KUKA KRL program: MyProgram_069().src

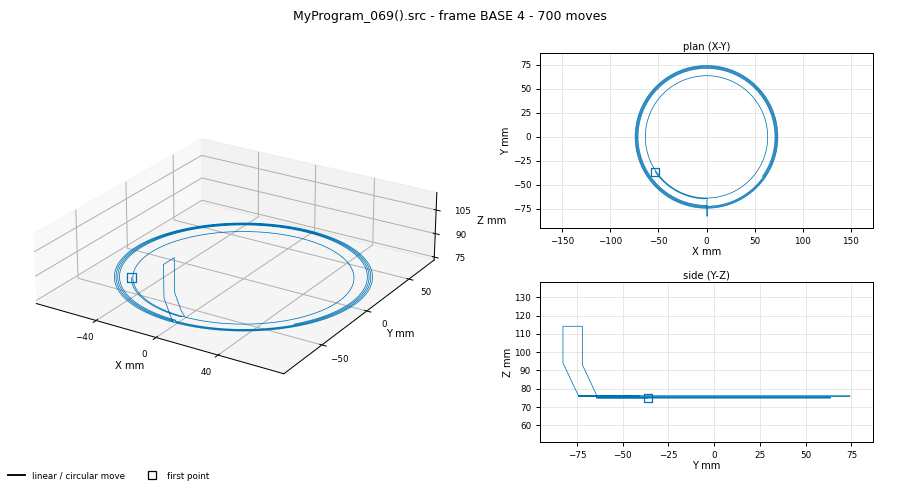
[picture p0: tool path of MyProgram_069().src in frame BASE 4, 700 of 700 moves have a stored position in this frame; points joined in program order, loops and branches not executed]
&ACCESS RVP
&REL 1
&PARAM TEMPLATE = C:\KRC\Roboter\Template\vorgabe
&PARAM EDITMASK = *
DEF MyProgram_069()
; ---- Setting reference (Base) ----
$BASE = BASE_DATA[4]

; --------------------------
; ---- Setting tool (TCP) ----
$TOOL = TOOL_DATA[3]
; --------------------------

$VEL.CP = VEL_APROX_PRINT
Startdeposition()
$VEL.CP = VEL_PRINT
LIN {X -53.2736,Y -36.3857,Z 75,A -150.3803,B 24.8918,C -2.4023,E1 24.8694,E2 -125.5307} C_DIS
LIN {X -51.112,Y -39.3636,Z 75,A -147.7583,B 24.8936,C -2.3813,E1 24.8737,E2 -128.1152} C_DIS
LIN {X -49.4525,Y -41.43,Z 75,A -144.3336,B 24.8921,C -2.3979,E1 24.8799,E2 -131.5953} C_DIS
LIN {X -46.3505,Y -44.8729,Z 75,A -140.9445,B 24.8943,C -2.3739,E1 24.8863,E2 -134.942} C_DIS
LIN {X -44.9329,Y -46.2927,Z 75,A -138.7085,B 24.8937,C -2.3797,E1 24.8908,E2 -137.2012} C_DIS
LIN {X -41.3789,Y -49.495,Z 75,A -134.5886,B 24.8947,C -2.3689,E1 24.8995,E2 -141.3115} C_DIS
LIN {X -38.5752,Y -51.7101,Z 75,A -131.7311,B 24.8958,C -2.3566,E1 24.9058,E2 -144.1501} C_DIS
LIN {X -36.3603,Y -53.2908,Z 75,A -129.2902,B 24.8961,C -2.3532,E1 24.9113,E2 -146.5913} C_DIS
LIN {X -34.0806,Y -54.7764,Z 75,A -126.7495,B 24.8961,C -2.3522,E1 24.9174,E2 -149.1377} C_DIS
LIN {X -31.5265,Y -56.2851,Z 75,A -124.1519,B 24.8966,C -2.3478,E1 24.9236,E2 -151.7325} C_DIS
LIN {X -29.0657,Y -57.5953,Z 75,A -121.6814,B 24.8969,C -2.3445,E1 24.9298,E2 -154.202} C_DIS
LIN {X -26.5923,Y -58.7774,Z 75,A -118.8897,B 24.8964,C -2.3496,E1 24.9369,E2 -157.0127} C_DIS
LIN {X -23.076,Y -60.2452,Z 75,A -115.9709,B 24.8976,C -2.3361,E1 24.9444,E2 -159.9057} C_DIS
LIN {X -20.7754,Y -61.0765,Z 75,A -113.7684,B 24.8977,C -2.335,E1 24.9502,E2 -162.1098} C_DIS
LIN {X -18.3054,Y -61.8615,Z 75,A -111.6866,B 24.8983,C -2.3285,E1 24.9557,E2 -164.1797} C_DIS
LIN {X -16.0814,Y -62.4765,Z 75,A -109.3686,B 24.8979,C -2.3332,E1 24.962,E2 -166.5126} C_DIS
LIN {X -13.5706,Y -63.0698,Z 75,A -107.0172,B 24.8979,C -2.3335,E1 24.9684,E2 -168.8676} C_DIS
LIN {X -10.8355,Y -63.5969,Z 75,A -104.5216,B 24.8979,C -2.3331,E1 24.9753,E2 -171.3649} C_DIS
LIN {X -7.9994,Y -64.0158,Z 75,A -102.109,B 24.8982,C -2.3296,E1 24.9819,E2 -173.771} C_DIS
LIN {X -4.131,Y -64.381,Z 75,A -98.8452,B 24.8986,C -2.3252,E1 24.991,E2 -177.0258} C_DIS
LIN {X -2.1333,Y -64.4779,Z 75,A -96.0689,B 24.8965,C -2.3486,E1 24.9989,E2 -179.8581} C_DIS
LIN {X -2.1333,Y -64.4779,Z 75,A -96.0689,B 24.8965,C -2.3486,E1 24.9989,E2 -179.8581} C_DIS
Enddeposition()
LIN {X 0.4536,Y -63.6088,Z 75,A -94.8897,B 24.8974,C -2.3386,E1 25.0022,E2 -181.0136} C_DIS
Startdeposition()
$VEL.CP = VEL_PRINT
LIN {X -1.5862,Y -63.5949,Z 75,A -97.6108,B 24.8992,C -2.3183,E1 24.9944,E2 -178.2442} C_DIS
LIN {X -4.665,Y -63.4434,Z 75,A -100.413,B 24.8992,C -2.3176,E1 24.9866,E2 -175.4395} C_DIS
LIN {X -7.7944,Y -63.1354,Z 75,A -103.2285,B 24.8992,C -2.3183,E1 24.9788,E2 -172.6239} C_DIS
LIN {X -10.8862,Y -62.6763,Z 75,A -106.0478,B 24.8991,C -2.319,E1 24.971,E2 -169.8036} C_DIS
LIN {X -13.9401,Y -62.0686,Z 75,A -108.8562,B 24.8991,C -2.3201,E1 24.9633,E2 -166.9946} C_DIS
LIN {X -16.9609,Y -61.312,Z 75,A -111.6742,B 24.8989,C -2.3215,E1 24.9557,E2 -164.1756} C_DIS
LIN {X -19.9607,Y -60.402,Z 75,A -114.4932,B 24.8987,C -2.3237,E1 24.9482,E2 -161.3568} C_DIS
LIN {X -22.895,Y -59.352,Z 75,A -117.3072,B 24.8985,C -2.326,E1 24.9408,E2 -158.5426} C_DIS
LIN {X -25.7932,Y -58.151,Z 75,A -120.1357,B 24.8982,C -2.3289,E1 24.9336,E2 -155.7143} C_DIS
LIN {X -28.6026,Y -56.8219,Z 75,A -122.9457,B 24.898,C -2.332,E1 24.9265,E2 -152.9043} C_DIS
LIN {X -31.3638,Y -55.3457,Z 75,A -125.7172,B 24.8975,C -2.3367,E1 24.9197,E2 -150.1363} C_DIS
LIN {X -33.5624,Y -54.0396,Z 75,A -128.0227,B 24.8973,C -2.34,E1 24.9143,E2 -147.8315} C_DIS
LIN {X -36.0815,Y -52.3917,Z 75,A -130.7821,B 24.897,C -2.3433,E1 24.9078,E2 -145.0708} C_DIS
LIN {X -38.5515,Y -50.6023,Z 75,A -133.5526,B 24.8966,C -2.3475,E1 24.9016,E2 -142.3004} C_DIS
LIN {X -40.9565,Y -48.6766,Z 75,A -136.3489,B 24.8962,C -2.3522,E1 24.8956,E2 -139.5047} C_DIS
LIN {X -43.2647,Y -46.6366,Z 75,A -139.132,B 24.8957,C -2.3574,E1 24.8898,E2 -136.7229} C_DIS
LIN {X -45.4504,Y -44.5087,Z 75,A -141.8393,B 24.8951,C -2.3639,E1 24.8845,E2 -134.0197} C_DIS
LIN {X -47.4246,Y -42.3981,Z 75,A -144.3013,B 24.8944,C -2.3724,E1 24.8799,E2 -131.567} C_DIS
LIN {X -49.1892,Y -40.3391,Z 75,A -146.9641,B 24.8943,C -2.3736,E1 24.8751,E2 -128.8949} C_DIS
LIN {X -51.0948,Y -37.8967,Z 75,A -149.7751,B 24.8937,C -2.3799,E1 24.8703,E2 -126.0854} C_DIS
LIN {X -52.8961,Y -35.339,Z 75,A -152.6098,B 24.8931,C -2.3865,E1 24.8658,E2 -123.2525} C_DIS
LIN {X -54.5639,Y -32.7051,Z 75,A -155.4478,B 24.8925,C -2.3932,E1 24.8617,E2 -120.416} C_DIS
LIN {X -56.1094,Y -29.9761,Z 75,A -158.2749,B 24.8918,C -2.4007,E1 24.8579,E2 -117.5918} C_DIS
LIN {X -57.5088,Y -27.1951,Z 75,A -161.0971,B 24.8912,C -2.408,E1 24.8544,E2 -114.7719} C_DIS
LIN {X -58.7706,Y -24.3485,Z 75,A -163.9365,B 24.8905,C -2.4153,E1 24.8513,E2 -111.9341} C_DIS
LIN {X -59.8972,Y -21.4281,Z 75,A -166.7555,B 24.8898,C -2.4234,E1 24.8486,E2 -109.1187} C_DIS
LIN {X -60.8747,Y -18.4692,Z 75,A -169.5856,B 24.8891,C -2.4313,E1 24.8462,E2 -106.291} C_DIS
LIN {X -61.7097,Y -15.4515,Z 75,A -172.4241,B 24.8883,C -2.4394,E1 24.8441,E2 -103.4554} C_DIS
LIN {X -62.3925,Y -12.4103,Z 75,A -175.2521,B 24.8876,C -2.4475,E1 24.8425,E2 -100.6303} C_DIS
LIN {X -62.9255,Y -9.3393,Z 75,A -178.0797,B 24.8868,C -2.4558,E1 24.8413,E2 -97.8057} C_DIS
LIN {X -63.3083,Y -6.237,Z 75,A 179.0777,B 24.886,C -2.4641,E1 24.8404,E2 -94.9658} C_DIS
LIN {X -63.5384,Y -3.1165,Z 75,A 176.2485,B 24.8852,C -2.4727,E1 24.8399,E2 -92.1403} C_DIS
LIN {X -63.6159,Y -0.0035,Z 75,A 173.3835,B 24.8845,C -2.4805,E1 24.8398,E2 -89.2765} C_DIS
LIN {X -63.5377,Y 3.1302,Z 75,A 170.5787,B 24.8836,C -2.4898,E1 24.8401,E2 -86.4771} C_DIS
LIN {X -63.3082,Y 6.2374,Z 75,A 167.7516,B 24.8828,C -2.4983,E1 24.8408,E2 -83.6533} C_DIS
LIN {X -62.9269,Y 9.3298,Z 75,A 164.9241,B 24.882,C -2.5067,E1 24.8418,E2 -80.8291} C_DIS
LIN {X -62.3946,Y 12.3995,Z 75,A 162.0978,B 24.8813,C -2.5152,E1 24.8433,E2 -78.0062} C_DIS
LIN {X -61.7084,Y 15.4568,Z 75,A 159.2405,B 24.8805,C -2.5233,E1 24.8451,E2 -75.1517} C_DIS
LIN {X -60.8705,Y 18.4828,Z 75,A 156.41,B 24.8796,C -2.532,E1 24.8473,E2 -72.3256} C_DIS
LIN {X -59.894,Y 21.4369,Z 75,A 153.5875,B 24.8789,C -2.5402,E1 24.8498,E2 -69.5067} C_DIS
LIN {X -58.774,Y 24.3404,Z 75,A 150.763,B 24.8781,C -2.5483,E1 24.8528,E2 -66.6855} C_DIS
LIN {X -57.5134,Y 27.1852,Z 75,A 147.9417,B 24.8773,C -2.5562,E1 24.856,E2 -63.8678} C_DIS
LIN {X -56.2186,Y 29.7687,Z 75,A 145.5305,B 24.8763,C -2.5674,E1 24.8591,E2 -61.4704} C_DIS
LIN {X -54.9606,Y 32.0339,Z 75,A 142.9607,B 24.876,C -2.5695,E1 24.8627,E2 -58.8924} C_DIS
LIN {X -53.3179,Y 34.6991,Z 75,A 140.1379,B 24.8753,C -2.5773,E1 24.8669,E2 -56.0738} C_DIS
LIN {X -51.5598,Y 37.2616,Z 75,A 137.3184,B 24.8746,C -2.5845,E1 24.8714,E2 -53.2575} C_DIS
LIN {X -49.8386,Y 39.5325,Z 75,A 134.7611,B 24.8739,C -2.5914,E1 24.8758,E2 -50.7046} C_DIS
LIN {X -47.895,Y 41.866,Z 75,A 131.9989,B 24.8733,C -2.5978,E1 24.8808,E2 -47.9451} C_DIS
LIN {X -45.8014,Y 44.1466,Z 75,A 129.1848,B 24.8727,C -2.6041,E1 24.8861,E2 -45.1338} C_DIS
LIN {X -43.5781,Y 46.3427,Z 75,A 126.4974,B 24.8718,C -2.6131,E1 24.8915,E2 -42.4568} C_DIS
LIN {X -41.5304,Y 48.1876,Z 75,A 123.8613,B 24.8715,C -2.6157,E1 24.897,E2 -39.8163} C_DIS
LIN {X -39.1322,Y 50.1548,Z 75,A 121.052,B 24.871,C -2.6213,E1 24.9032,E2 -37.0101} C_DIS
LIN {X -36.6395,Y 52.0036,Z 75,A 118.2409,B 24.8705,C -2.6266,E1 24.9095,E2 -34.2018} C_DIS
LIN {X -34.0348,Y 53.7445,Z 75,A 115.4063,B 24.87,C -2.6317,E1 24.9161,E2 -31.3701} C_DIS
LIN {X -31.3169,Y 55.372,Z 75,A 112.5717,B 24.8694,C -2.6371,E1 24.923,E2 -28.5398} C_DIS
LIN {X -28.5819,Y 56.8322,Z 75,A 109.7423,B 24.869,C -2.6409,E1 24.93,E2 -25.7118} C_DIS
LIN {X -25.7746,Y 58.1593,Z 75,A 106.934,B 24.8686,C -2.6449,E1 24.9371,E2 -22.9059} C_DIS
LIN {X -22.9048,Y 59.3481,Z 75,A 104.1261,B 24.8683,C -2.6484,E1 24.9444,E2 -20.1004} C_DIS
LIN {X -19.9491,Y 60.4059,Z 75,A 101.3458,B 24.8679,C -2.6528,E1 24.9517,E2 -17.3253} C_DIS
LIN {X -17.5047,Y 61.158,Z 75,A 99.0947,B 24.8675,C -2.6564,E1 24.9577,E2 -15.0789} C_DIS
LIN {X -14.6786,Y 61.898,Z 75,A 96.3519,B 24.8675,C -2.6566,E1 24.9651,E2 -12.3326} C_DIS
LIN {X -11.6341,Y 62.5418,Z 75,A 93.5368,B 24.8673,C -2.6586,E1 24.9729,E2 -9.5191} C_DIS
LIN {X -9.1143,Y 62.9575,Z 75,A 91.3179,B 24.8669,C -2.6619,E1 24.979,E2 -7.3062} C_DIS
LIN {X -6.1891,Y 63.3127,Z 75,A 88.5793,B 24.8669,C -2.6615,E1 24.9866,E2 -4.5649} C_DIS
LIN {X -3.0984,Y 63.5392,Z 75,A 85.7848,B 24.8669,C -2.6625,E1 24.9944,E2 -1.772} C_DIS
LIN {X 0.0032,Y 63.6148,Z 75,A 82.9856,B 24.8669,C -2.6631,E1 25.0022,E2 1.026} C_DIS
LIN {X 3.1338,Y 63.5375,Z 75,A 80.1649,B 24.8669,C -2.6633,E1 25.01,E2 3.8456} C_DIS
LIN {X 6.2357,Y 63.3084,Z 75,A 77.3535,B 24.8669,C -2.6629,E1 25.0179,E2 6.6563} C_DIS
LIN {X 9.3404,Y 62.9253,Z 75,A 74.5461,B 24.8669,C -2.6624,E1 25.0256,E2 9.4624} C_DIS
LIN {X 12.4092,Y 62.3927,Z 75,A 71.7413,B 24.8669,C -2.6614,E1 25.0333,E2 12.2666} C_DIS
LIN {X 15.4667,Y 61.7059,Z 75,A 68.9232,B 24.8671,C -2.6599,E1 25.041,E2 15.0841} C_DIS
LIN {X 18.47,Y 60.8744,Z 75,A 66.1206,B 24.8673,C -2.6581,E1 25.0485,E2 17.8864} C_DIS
LIN {X 21.4292,Y 59.8968,Z 75,A 63.3044,B 24.8676,C -2.6555,E1 25.0559,E2 20.7031} C_DIS
LIN {X 24.3533,Y 58.7686,Z 75,A 60.5053,B 24.8678,C -2.6533,E1 25.0632,E2 23.5012} C_DIS
LIN {X 27.1924,Y 57.5101,Z 75,A 57.7015,B 24.8681,C -2.6499,E1 25.0703,E2 26.3058} C_DIS
LIN {X 29.9949,Y 56.0994,Z 75,A 54.8938,B 24.8685,C -2.6467,E1 25.0773,E2 29.1134} C_DIS
LIN {X 32.706,Y 54.5633,Z 75,A 52.0953,B 24.8688,C -2.6429,E1 25.084,E2 31.9123} C_DIS
LIN {X 35.3388,Y 52.8962,Z 75,A 49.3009,B 24.8692,C -2.6389,E1 25.0906,E2 34.7072} C_DIS
LIN {X 37.8864,Y 51.1024,Z 75,A 46.4928,B 24.8697,C -2.6341,E1 25.0969,E2 37.5168} C_DIS
LIN {X 40.3605,Y 49.1718,Z 75,A 43.6883,B 24.8702,C -2.6294,E1 25.103,E2 40.3217} C_DIS
LIN {X 42.7186,Y 47.1377,Z 75,A 40.8915,B 24.8707,C -2.6242,E1 25.1089,E2 43.12} C_DIS
LIN {X 44.9873,Y 44.9775,Z 75,A 38.0869,B 24.8712,C -2.6188,E1 25.1145,E2 45.9256} C_DIS
LIN {X 47.1345,Y 42.7221,Z 75,A 35.2939,B 24.8718,C -2.6129,E1 25.1198,E2 48.7202} C_DIS
LIN {X 49.1744,Y 40.3574,Z 75,A 32.4874,B 24.8724,C -2.6066,E1 25.1249,E2 51.5287} C_DIS
LIN {X 51.1003,Y 37.8892,Z 75,A 29.6918,B 24.873,C -2.6005,E1 25.1296,E2 54.3256} C_DIS
LIN {X 52.8943,Y 35.3417,Z 75,A 27.0861,B 24.8732,C -2.5984,E1 25.1337,E2 56.9234} C_DIS
LIN {X 54.1864,Y 33.3262,Z 75,A 24.7652,B 24.8742,C -2.5888,E1 25.1372,E2 59.2552} C_DIS
LIN {X 55.742,Y 30.6537,Z 75,A 21.9932,B 24.8749,C -2.5818,E1 25.141,E2 62.0296} C_DIS
LIN {X 57.1695,Y 27.9014,Z 75,A 19.2132,B 24.8756,C -2.5744,E1 25.1445,E2 64.8121} C_DIS
LIN {X 58.4611,Y 25.0825,Z 75,A 16.4284,B 24.8763,C -2.5668,E1 25.1476,E2 67.5998} C_DIS
LIN {X 59.6287,Y 22.1644,Z 75,A 13.623,B 24.877,C -2.5593,E1 25.1505,E2 70.4073} C_DIS
LIN {X 60.6496,Y 19.1951,Z 75,A 10.8159,B 24.8778,C -2.5515,E1 25.1529,E2 73.217} C_DIS
LIN {X 61.5159,Y 16.2058,Z 75,A 8.0311,B 24.8785,C -2.5436,E1 25.155,E2 76.0046} C_DIS
LIN {X 62.2351,Y 13.1768,Z 75,A 5.2439,B 24.8793,C -2.5354,E1 25.1567,E2 78.7948} C_DIS
LIN {X 62.8086,Y 10.0955,Z 75,A 2.6298,B 24.8797,C -2.532,E1 25.158,E2 81.4017} C_DIS
LIN {X 63.1502,Y 7.6694,Z 75,A 0.2777,B 24.8807,C -2.5215,E1 25.1588,E2 83.7648} C_DIS
LIN {X 63.4448,Y 4.6442,Z 75,A -2.4543,B 24.8815,C -2.513,E1 25.1595,E2 86.5005} C_DIS
LIN {X 63.5907,Y 1.723,Z 75,A -5.0784,B 24.8822,C -2.505,E1 25.1598,E2 89.128} C_DIS
LIN {X 63.5948,Y -1.5886,Z 75,A -8.0424,B 24.8831,C -2.496,E1 25.1597,E2 92.0957} C_DIS
LIN {X 63.4416,Y -4.6895,Z 75,A -10.82,B 24.8838,C -2.4876,E1 25.1592,E2 94.8766} C_DIS
LIN {X 63.1371,Y -7.7813,Z 75,A -13.6018,B 24.8846,C -2.4791,E1 25.1583,E2 97.6619} C_DIS
LIN {X 62.6766,Y -10.885,Z 75,A -16.4077,B 24.8854,C -2.4707,E1 25.1571,E2 100.4712} C_DIS
LIN {X 62.0686,Y -13.9403,Z 75,A -19.1944,B 24.8862,C -2.4624,E1 25.1555,E2 103.2614} C_DIS
LIN {X 61.3116,Y -16.9624,Z 75,A -21.9821,B 24.887,C -2.4541,E1 25.1535,E2 106.0527} C_DIS
LIN {X 60.4077,Y -19.9434,Z 75,A -24.7683,B 24.8877,C -2.4459,E1 25.1512,E2 108.8423} C_DIS
LIN {X 59.3578,Y -22.8796,Z 75,A -27.5816,B 24.8885,C -2.4373,E1 25.1484,E2 111.6604} C_DIS
LIN {X 58.1492,Y -25.7973,Z 75,A -30.3781,B 24.8892,C -2.4299,E1 25.1453,E2 114.4589} C_DIS
LIN {X 56.8221,Y -28.6023,Z 75,A -33.159,B 24.8899,C -2.4221,E1 25.1419,E2 117.2435} C_DIS
LIN {X 55.3471,Y -31.3614,Z 75,A -35.9584,B 24.8906,C -2.4144,E1 25.1382,E2 120.0464} C_DIS
LIN {X 53.7461,Y -34.0323,Z 75,A -38.7473,B 24.8913,C -2.4069,E1 25.1341,E2 122.8388} C_DIS
LIN {X 52.3355,Y -36.1624,Z 75,A -40.9259,B 24.8916,C -2.4037,E1 25.1307,E2 125.0143} C_DIS
LIN {X 50.616,Y -38.5337,Z 75,A -43.653,B 24.8924,C -2.3944,E1 25.1261,E2 127.7503} C_DIS
LIN {X 48.6741,Y -40.9594,Z 75,A -46.4378,B 24.893,C -2.3875,E1 25.1212,E2 130.5385} C_DIS
LIN {X 46.6155,Y -43.2878,Z 75,A -49.2468,B 24.8937,C -2.3802,E1 25.1159,E2 133.3523} C_DIS
LIN {X 44.4109,Y -45.5466,Z 75,A -52.0468,B 24.8942,C -2.3745,E1 25.1104,E2 136.154} C_DIS
LIN {X 42.1345,Y -47.6605,Z 75,A -54.8314,B 24.8947,C -2.3684,E1 25.1046,E2 138.9419} C_DIS
LIN {X 39.7565,Y -49.6614,Z 75,A -57.6197,B 24.8953,C -2.3625,E1 25.0986,E2 141.7334} C_DIS
LIN {X 37.2535,Y -51.5656,Z 75,A -60.4288,B 24.8957,C -2.3572,E1 25.0923,E2 144.5449} C_DIS
LIN {X 34.6862,Y -53.3264,Z 75,A -63.2303,B 24.8962,C -2.3518,E1 25.0858,E2 147.3498} C_DIS
LIN {X 32.0353,Y -54.9598,Z 75,A -66.0387,B 24.8967,C -2.3466,E1 25.079,E2 150.162} C_DIS
LIN {X 29.2897,Y -56.4708,Z 75,A -68.8327,B 24.897,C -2.3425,E1 25.0721,E2 152.9576} C_DIS
LIN {X 26.5014,Y -57.8317,Z 75,A -71.621,B 24.8974,C -2.3383,E1 25.0651,E2 155.7487} C_DIS
LIN {X 23.8555,Y -58.9714,Z 75,A -73.967,B 24.8972,C -2.3405,E1 25.0591,E2 158.0841} C_DIS
LIN {X 21.4149,Y -59.9018,Z 75,A -76.5529,B 24.898,C -2.3319,E1 25.0523,E2 160.685} C_DIS
LIN {X 18.4567,Y -60.8784,Z 75,A -79.3518,B 24.8982,C -2.3287,E1 25.0448,E2 163.4861} C_DIS
LIN {X 15.4544,Y -61.709,Z 75,A -81.9653,B 24.8982,C -2.3303,E1 25.0378,E2 166.0918} C_DIS
LIN {X 13.1313,Y -62.2445,Z 75,A -84.2896,B 24.8986,C -2.3243,E1 25.0314,E2 168.4273} C_DIS
LIN {X 10.0828,Y -62.8105,Z 75,A -87.0793,B 24.8988,C -2.3222,E1 25.0237,E2 171.219} C_DIS
LIN {X 7.0055,Y -63.2278,Z 75,A -89.8194,B 24.8988,C -2.3217,E1 25.0161,E2 173.958} C_DIS
LIN {X 4.4282,Y -63.4594,Z 75,A -92.137,B 24.8989,C -2.3209,E1 25.0097,E2 176.2763} C_DIS
LIN {X 1.4801,Y -63.5971,Z 75,A -94.8431,B 24.8991,C -2.319,E1 25.0021,E2 178.9864} C_DIS
LIN {X 1.4801,Y -63.5971,Z 75,A -94.8431,B 24.8991,C -2.319,E1 25.0021,E2 178.9864} C_DIS
Enddeposition()
LIN {X 0.4776,Y -65.7217,Z 79.5315,A -94.88,B 24.8977,C -2.3345,E1 25.0021,E2 178.9864} C_DIS
LIN {X 0.5496,Y -72.0606,Z 93.1262,A -94.8556,B 24.8986,C -2.3242,E1 25.0021,E2 178.9864} C_DIS
LIN {X 0.5496,Y -72.0606,Z 114.1262,A -95.2134,B 24.885,C -2.4748,E1 25.0021,E2 178.9864} C_DIS
LIN {X 0.6266,Y -82.6562,Z 114.1262,A -94.6615,B 24.9002,C -2.3061,E1 25.0026,E2 178.8353} C_DIS
LIN {X 0.6266,Y -82.6562,Z 94.1262,A -94.3209,B 24.9123,C -2.1627,E1 25.0026,E2 178.8353} C_DIS
LIN {X 0.5379,Y -76.3176,Z 80.5315,A -94.3434,B 24.9115,C -2.1722,E1 25.0026,E2 178.8353} C_DIS
LIN {X 0.5083,Y -74.2047,Z 76,A -94.3524,B 24.9112,C -2.176,E1 25.0026,E2 178.8353} C_DIS
Startdeposition()
$VEL.CP = VEL_PRINT
LIN {X 3.1308,Y -74.1412,Z 76,A -92.2496,B 24.911,C -2.1787,E1 25.0084,E2 176.7265} C_DIS
LIN {X 5.9684,Y -73.9669,Z 76,A -90.1014,B 24.911,C -2.1785,E1 25.0144,E2 174.5799} C_DIS
LIN {X 8.5765,Y -73.71,Z 76,A -88.0356,B 24.9108,C -2.1808,E1 25.0202,E2 172.51} C_DIS
LIN {X 11.2837,Y -73.3444,Z 76,A -85.9296,B 24.9107,C -2.1821,E1 25.026,E2 170.4027} C_DIS
LIN {X 14.0849,Y -72.8583,Z 76,A -83.5817,B 24.9102,C -2.1881,E1 25.0325,E2 168.0433} C_DIS
LIN {X 17.1465,Y -72.2006,Z 76,A -81.2572,B 24.9102,C -2.1877,E1 25.0388,E2 165.7228} C_DIS
LIN {X 19.9124,Y -71.4865,Z 76,A -79.0131,B 24.9099,C -2.1911,E1 25.0449,E2 163.4742} C_DIS
LIN {X 22.8976,Y -70.5863,Z 76,A -76.5668,B 24.9096,C -2.195,E1 25.0514,E2 161.0231} C_DIS
LIN {X 25.8557,Y -69.5587,Z 76,A -74.2082,B 24.9096,C -2.1965,E1 25.0576,E2 158.666} C_DIS
LIN {X 28.7668,Y -68.4046,Z 76,A -71.9018,B 24.9095,C -2.1968,E1 25.0635,E2 156.3641} C_DIS
LIN {X 31.3659,Y -67.2525,Z 76,A -69.5577,B 24.9089,C -2.2043,E1 25.0695,E2 154.008} C_DIS
LIN {X 34.176,Y -65.8705,Z 76,A -67.2009,B 24.9087,C -2.2065,E1 25.0754,E2 151.6524} C_DIS
LIN {X 36.5773,Y -64.568,Z 76,A -65.0997,B 24.9084,C -2.21,E1 25.0805,E2 149.5492} C_DIS
LIN {X 38.9291,Y -63.1779,Z 76,A -62.999,B 24.9081,C -2.2136,E1 25.0855,E2 147.4465} C_DIS
LIN {X 41.5591,Y -61.4781,Z 76,A -60.6952,B 24.908,C -2.215,E1 25.0909,E2 145.1469} C_DIS
LIN {X 43.8835,Y -59.8411,Z 76,A -58.4277,B 24.9074,C -2.2216,E1 25.0961,E2 142.8718} C_DIS
LIN {X 46.37,Y -57.9375,Z 76,A -56.0355,B 24.907,C -2.226,E1 25.1013,E2 140.478} C_DIS
LIN {X 48.4711,Y -56.1914,Z 76,A -53.9365,B 24.9067,C -2.2304,E1 25.1058,E2 138.3768} C_DIS
LIN {X 50.5065,Y -54.3693,Z 76,A -51.8379,B 24.9063,C -2.235,E1 25.1101,E2 136.2759} C_DIS
LIN {X 52.4734,Y -52.4734,Z 76,A -49.704,B 24.9058,C -2.2407,E1 25.1144,E2 134.1373} C_DIS
LIN {X 54.6395,Y -50.2119,Z 76,A -47.4031,B 24.9056,C -2.2433,E1 25.1188,E2 131.8403} C_DIS
LIN {X 56.4507,Y -48.1668,Z 76,A -45.3057,B 24.9052,C -2.2483,E1 25.1226,E2 129.7405} C_DIS
LIN {X 58.2543,Y -45.9691,Z 76,A -43.0841,B 24.9046,C -2.2549,E1 25.1265,E2 127.514} C_DIS
LIN {X 59.8411,Y -43.8835,Z 76,A -41.1116,B 24.9043,C -2.2588,E1 25.1298,E2 125.5416} C_DIS
LIN {X 61.4781,Y -41.5591,Z 76,A -38.7739,B 24.9034,C -2.269,E1 25.1335,E2 123.1911} C_DIS
LIN {X 63.1779,Y -38.9291,Z 76,A -36.4588,B 24.9031,C -2.2727,E1 25.137,E2 120.879} C_DIS
LIN {X 64.568,Y -36.5773,Z 76,A -34.3629,B 24.9026,C -2.2784,E1 25.1399,E2 118.7806} C_DIS
LIN {X 65.8705,Y -34.176,Z 76,A -32.2314,B 24.902,C -2.2852,E1 25.1427,E2 116.6442} C_DIS
LIN {X 67.2525,Y -31.3659,Z 76,A -29.9329,B 24.9017,C -2.2888,E1 25.1455,E2 114.3496} C_DIS
LIN {X 68.4046,Y -28.7668,Z 76,A -27.5965,B 24.9008,C -2.2996,E1 25.1481,E2 112.0003} C_DIS
LIN {X 69.5587,Y -25.8557,Z 76,A -25.2469,B 24.9003,C -2.3049,E1 25.1504,E2 109.6513} C_DIS
LIN {X 70.5863,Y -22.8976,Z 76,A -22.9492,B 24.9,C -2.3088,E1 25.1525,E2 107.3575} C_DIS
LIN {X 71.3812,Y -20.284,Z 76,A -20.8543,B 24.8995,C -2.3149,E1 25.1541,E2 105.26} C_DIS
LIN {X 72.1058,Y -17.5349,Z 76,A -18.719,B 24.899,C -2.32,E1 25.1556,E2 103.125} C_DIS
LIN {X 72.68,Y -14.9779,Z 76,A -16.665,B 24.8984,C -2.3273,E1 25.1568,E2 101.0657} C_DIS
LIN {X 73.182,Y -12.2926,Z 76,A -14.5704,B 24.8978,C -2.3336,E1 25.1578,E2 98.9687} C_DIS
LIN {X 73.5992,Y -9.4804,Z 76,A -12.235,B 24.8968,C -2.3447,E1 25.1587,E2 96.6207} C_DIS
LIN {X 73.935,Y -6.3669,Z 76,A -9.8862,B 24.8963,C -2.3503,E1 25.1593,E2 94.2725} C_DIS
LIN {X 74.1193,Y -3.6412,Z 76,A -7.8274,B 24.8959,C -2.3555,E1 25.1597,E2 92.2137} C_DIS
LIN {X 74.1957,Y -1.3103,Z 76,A -6.1475,B 24.8957,C -2.3577,E1 25.1597,E2 90.5387} C_DIS
LIN {X 74.1957,Y 1.3103,Z 76,A -4.0981,B 24.8951,C -2.3649,E1 25.1597,E2 88.4846} C_DIS
LIN {X 74.0911,Y 4.1514,Z 76,A -1.9627,B 24.8946,C -2.37,E1 25.1595,E2 86.3496} C_DIS
LIN {X 73.8983,Y 6.765,Z 76,A 0.0911,B 24.8939,C -2.3773,E1 25.159,E2 84.2908} C_DIS
LIN {X 73.5849,Y 9.5906,Z 76,A 2.4272,B 24.893,C -2.3884,E1 25.1582,E2 81.9424} C_DIS
LIN {X 73.1161,Y 12.6868,Z 76,A 4.7405,B 24.8926,C -2.3927,E1 25.1572,E2 79.6324} C_DIS
LIN {X 72.5996,Y 15.3695,Z 76,A 6.8712,B 24.8919,C -2.3998,E1 25.156,E2 77.4973} C_DIS
LIN {X 71.8852,Y 18.4184,Z 76,A 9.1691,B 24.8916,C -2.4036,E1 25.1544,E2 75.2037} C_DIS
LIN {X 71.1269,Y 21.1584,Z 76,A 11.3053,B 24.8911,C -2.4085,E1 25.1528,E2 73.0683} C_DIS
LIN {X 70.3355,Y 23.6567,Z 76,A 13.3602,B 24.8905,C -2.4154,E1 25.151,E2 71.0087} C_DIS
LIN {X 69.3777,Y 26.3335,Z 76,A 15.4966,B 24.8901,C -2.42,E1 25.149,E2 68.8734} C_DIS
LIN {X 68.4046,Y 28.7668,Z 76,A 17.552,B 24.8895,C -2.4268,E1 25.1468,E2 66.8134} C_DIS
LIN {X 67.2525,Y 31.3659,Z 76,A 19.8894,B 24.8885,C -2.4371,E1 25.1441,E2 64.4642} C_DIS
LIN {X 65.8705,Y 34.176,Z 76,A 22.2404,B 24.8881,C -2.4417,E1 25.1411,E2 62.1147} C_DIS
LIN {X 64.568,Y 36.5773,Z 76,A 24.3373,B 24.8876,C -2.447,E1 25.1382,E2 60.0162} C_DIS
LIN {X 62.9661,Y 39.2681,Z 76,A 26.6375,B 24.8874,C -2.4499,E1 25.1349,E2 57.721} C_DIS
LIN {X 61.4158,Y 41.6512,Z 76,A 28.7758,B 24.887,C -2.4538,E1 25.1316,E2 55.5841} C_DIS
LIN {X 59.8411,Y 43.8835,Z 76,A 31.0743,B 24.886,C -2.4645,E1 25.1278,E2 53.2715} C_DIS
LIN {X 57.9375,Y 46.37,Z 76,A 33.4848,B 24.8855,C -2.47,E1 25.1237,E2 50.8593} C_DIS
LIN {X 55.9285,Y 48.7722,Z 76,A 35.7291,B 24.8855,C -2.4705,E1 25.1196,E2 48.624} C_DIS
LIN {X 54.0954,Y 50.7977,Z 76,A 37.8282,B 24.885,C -2.4749,E1 25.1157,E2 46.5238} C_DIS
LIN {X 52.189,Y 52.7544,Z 76,A 39.9276,B 24.8847,C -2.479,E1 25.1115,E2 44.4234} C_DIS
LIN {X 50.13,Y 54.7147,Z 76,A 42.0684,B 24.8844,C -2.4819,E1 25.1072,E2 42.2846} C_DIS
LIN {X 48.1668,Y 56.4507,Z 76,A 44.1279,B 24.8839,C -2.4868,E1 25.1028,E2 40.2215} C_DIS
LIN {X 45.7939,Y 58.3927,Z 76,A 46.6185,B 24.8832,C -2.4947,E1 25.0974,E2 37.7218} C_DIS
LIN {X 43.4713,Y 60.1429,Z 76,A 48.791,B 24.883,C -2.4964,E1 25.0925,E2 35.5528} C_DIS
LIN {X 41.2281,Y 61.7022,Z 76,A 50.9286,B 24.8826,C -2.5006,E1 25.0876,E2 33.4125} C_DIS
LIN {X 38.5875,Y 63.3855,Z 76,A 53.2343,B 24.8826,C -2.5012,E1 25.0821,E2 31.1128} C_DIS
LIN {X 36.2283,Y 64.7629,Z 76,A 55.3372,B 24.8823,C -2.504,E1 25.077,E2 29.0096} C_DIS
LIN {X 33.82,Y 66.0525,Z 76,A 57.4404,B 24.8821,C -2.5065,E1 25.0718,E2 26.9062} C_DIS
LIN {X 31.1818,Y 67.3382,Z 76,A 59.6237,B 24.8821,C -2.5069,E1 25.0663,E2 24.7276} C_DIS
LIN {X 28.7668,Y 68.4046,Z 76,A 61.8908,B 24.8812,C -2.5154,E1 25.0605,E2 22.4458} C_DIS
LIN {X 25.8557,Y 69.5587,Z 76,A 64.2513,B 24.8812,C -2.5161,E1 25.0543,E2 20.0888} C_DIS
LIN {X 22.8976,Y 70.5863,Z 76,A 66.5602,B 24.8812,C -2.5152,E1 25.0482,E2 17.7866} C_DIS
LIN {X 20.284,Y 71.3812,Z 76,A 68.6666,B 24.8812,C -2.5166,E1 25.0426,E2 15.6806} C_DIS
LIN {X 17.6429,Y 72.0795,Z 76,A 70.7733,B 24.881,C -2.5178,E1 25.0369,E2 13.5742} C_DIS
LIN {X 14.9779,Y 72.68,Z 76,A 72.8802,B 24.881,C -2.5187,E1 25.0311,E2 11.4678} C_DIS
LIN {X 12.2072,Y 73.1963,Z 76,A 75.0193,B 24.881,C -2.5185,E1 25.0253,E2 9.3315} C_DIS
LIN {X 9.4804,Y 73.5992,Z 76,A 77.3387,B 24.8804,C -2.5241,E1 25.0188,E2 7.0008} C_DIS
LIN {X 6.3669,Y 73.935,Z 76,A 79.7037,B 24.8805,C -2.523,E1 25.0122,E2 4.64} C_DIS
LIN {X 3.6412,Y 74.1193,Z 76,A 81.7771,B 24.8806,C -2.522,E1 25.0065,E2 2.5697} C_DIS
LIN {X 0.9107,Y 74.2031,Z 76,A 83.8871,B 24.8806,C -2.5217,E1 25.0006,E2 0.4607} C_DIS
LIN {X -1.8314,Y 74.186,Z 76,A 85.9997,B 24.8806,C -2.5211,E1 24.9947,E2 -1.6505} C_DIS
LIN {X -4.5505,Y 74.069,Z 76,A 88.1446,B 24.8806,C -2.5215,E1 24.9887,E2 -3.797} C_DIS
LIN {X -7.3724,Y 73.841,Z 76,A 90.2413,B 24.881,C -2.5181,E1 24.9829,E2 -5.8867} C_DIS
LIN {X -9.9871,Y 73.5335,Z 76,A 92.3326,B 24.881,C -2.5184,E1 24.9771,E2 -7.9802} C_DIS
LIN {X -12.7637,Y 73.1023,Z 76,A 94.4986,B 24.881,C -2.5168,E1 24.9711,E2 -10.1444} C_DIS
LIN {X -15.76,Y 72.5144,Z 76,A 96.7993,B 24.8814,C -2.5134,E1 24.9649,E2 -12.4397} C_DIS
LIN {X -18.4184,Y 71.8852,Z 76,A 98.9131,B 24.8816,C -2.5115,E1 24.9591,E2 -14.552} C_DIS
LIN {X -21.1584,Y 71.1269,Z 76,A 101.1362,B 24.8818,C -2.5099,E1 24.9532,E2 -16.7749} C_DIS
LIN {X -23.762,Y 70.3,Z 76,A 103.1834,B 24.8821,C -2.5059,E1 24.9477,E2 -18.8162} C_DIS
LIN {X -26.3335,Y 69.3777,Z 76,A 105.5011,B 24.8819,C -2.5084,E1 24.9416,E2 -21.1447} C_DIS
LIN {X -29.2376,Y 68.2062,Z 76,A 107.838,B 24.8824,C -2.5029,E1 24.9356,E2 -23.474} C_DIS
LIN {X -31.7283,Y 67.0838,Z 76,A 110.0452,B 24.8824,C -2.5022,E1 24.93,E2 -25.6849} C_DIS
LIN {X -34.176,Y 65.8705,Z 76,A 112.0716,B 24.883,C -2.4967,E1 24.925,E2 -27.7036} C_DIS
LIN {X -36.5773,Y 64.568,Z 76,A 114.189,B 24.8833,C -2.4933,E1 24.9199,E2 -29.8191} C_DIS
LIN {X -38.9787,Y 63.1469,Z 76,A 116.3191,B 24.8837,C -2.4888,E1 24.9148,E2 -31.945} C_DIS
LIN {X -41.2281,Y 61.7022,Z 76,A 118.4253,B 24.884,C -2.4859,E1 24.9099,E2 -34.0513} C_DIS
LIN {X -43.4713,Y 60.1429,Z 76,A 120.5441,B 24.8844,C -2.482,E1 24.905,E2 -36.1678} C_DIS
LIN {X -45.6555,Y 58.5021,Z 76,A 122.6995,B 24.8847,C -2.4787,E1 24.9003,E2 -38.3232} C_DIS
LIN {X -47.7779,Y 56.782,Z 76,A 124.8191,B 24.8851,C -2.4743,E1 24.8957,E2 -40.4406} C_DIS
LIN {X -49.8355,Y 54.985,Z 76,A 126.9031,B 24.8856,C -2.469,E1 24.8914,E2 -42.5201} C_DIS
LIN {X -51.8256,Y 53.1134,Z 76,A 129.0597,B 24.8859,C -2.4652,E1 24.887,E2 -44.6765} C_DIS
LIN {X -53.7454,Y 51.1699,Z 76,A 131.1443,B 24.8865,C -2.4595,E1 24.883,E2 -46.7566} C_DIS
LIN {X -55.5924,Y 49.157,Z 76,A 133.3017,B 24.8868,C -2.4554,E1 24.879,E2 -48.9138} C_DIS
LIN {X -57.6158,Y 46.7669,Z 76,A 135.6287,B 24.8876,C -2.4471,E1 24.8748,E2 -51.2316} C_DIS
LIN {X -59.2981,Y 44.6145,Z 76,A 137.7504,B 24.8881,C -2.4418,E1 24.8712,E2 -53.3509} C_DIS
LIN {X -60.9,Y 42.4017,Z 76,A 139.8728,B 24.8886,C -2.4364,E1 24.8678,E2 -55.4708} C_DIS
LIN {X -62.4795,Y 40.0379,Z 76,A 142.0365,B 24.8892,C -2.4296,E1 24.8645,E2 -57.6291} C_DIS
LIN {X -63.8543,Y 37.8067,Z 76,A 144.1179,B 24.8896,C -2.4253,E1 24.8615,E2 -59.7109} C_DIS
LIN {X -65.2556,Y 35.3331,Z 76,A 146.2821,B 24.8903,C -2.4182,E1 24.8586,E2 -61.8697} C_DIS
LIN {X -66.5119,Y 32.9073,Z 76,A 148.4053,B 24.8908,C -2.4124,E1 24.8559,E2 -63.9903} C_DIS
LIN {X -67.678,Y 30.4369,Z 76,A 150.5288,B 24.8913,C -2.4065,E1 24.8534,E2 -66.1113} C_DIS
LIN {X -68.7525,Y 27.9252,Z 76,A 152.8558,B 24.8914,C -2.4052,E1 24.8509,E2 -68.4482} C_DIS
LIN {X -69.8707,Y 25.0001,Z 76,A 155.2371,B 24.8922,C -2.397,E1 24.8486,E2 -70.8233} C_DIS
LIN {X -70.8619,Y 22.0296,Z 76,A 157.5671,B 24.893,C -2.3875,E1 24.8466,E2 -73.144} C_DIS
LIN {X -71.6248,Y 19.4065,Z 76,A 159.691,B 24.8936,C -2.3813,E1 24.845,E2 -75.2655} C_DIS
LIN {X -72.2905,Y 16.757,Z 76,A 161.8153,B 24.8941,C -2.3751,E1 24.8436,E2 -77.3872} C_DIS
LIN {X -72.922,Y 13.7542,Z 76,A 164.2957,B 24.8946,C -2.3702,E1 24.8423,E2 -79.8706} C_DIS
LIN {X -73.4055,Y 10.8887,Z 76,A 166.5664,B 24.8952,C -2.3637,E1 24.8413,E2 -82.1393} C_DIS
LIN {X -73.7981,Y 7.7819,Z 76,A 168.8966,B 24.896,C -2.354,E1 24.8405,E2 -84.4603} C_DIS
LIN {X -74.042,Y 4.9494,Z 76,A 171.0624,B 24.8967,C -2.3464,E1 24.8401,E2 -86.6208} C_DIS
LIN {X -74.1793,Y 2.0496,Z 76,A 173.4782,B 24.897,C -2.3433,E1 24.8398,E2 -89.0439} C_DIS
LIN {X -74.2031,Y -0.9107,Z 76,A 175.7723,B 24.8976,C -2.3362,E1 24.8398,E2 -91.3348} C_DIS
LIN {X -74.1193,Y -3.6412,Z 76,A 177.8605,B 24.8982,C -2.3291,E1 24.8401,E2 -93.4185} C_DIS
LIN {X -73.935,Y -6.3669,Z 76,A -179.9791,B 24.8987,C -2.3236,E1 24.8405,E2 -95.579} C_DIS
LIN {X -73.5992,Y -9.4804,Z 76,A -177.6491,B 24.8995,C -2.314,E1 24.8413,E2 -97.9001} C_DIS
LIN {X -73.182,Y -12.2926,Z 76,A -175.4836,B 24.9002,C -2.3066,E1 24.8422,E2 -100.0605} C_DIS
LIN {X -72.68,Y -14.9779,Z 76,A -173.1566,B 24.9003,C -2.3052,E1 24.8435,E2 -102.3979} C_DIS
LIN {X -71.9847,Y -18.0312,Z 76,A -170.775,B 24.901,C -2.297,E1 24.845,E2 -104.7738} C_DIS
LIN {X -71.2722,Y -20.6686,Z 76,A -168.6379,B 24.9015,C -2.2913,E1 24.8467,E2 -106.9099} C_DIS
LIN {X -70.4632,Y -23.2779,Z 76,A -166.5641,B 24.9021,C -2.2842,E1 24.8484,E2 -108.9787} C_DIS
LIN {X -69.5587,Y -25.8557,Z 76,A -164.4049,B 24.9025,C -2.2793,E1 24.8505,E2 -111.1383} C_DIS
LIN {X -68.4046,Y -28.7668,Z 76,A -162.0764,B 24.9033,C -2.2703,E1 24.8529,E2 -113.4583} C_DIS
LIN {X -67.2525,Y -31.3659,Z 76,A -159.7094,B 24.9035,C -2.2682,E1 24.8557,E2 -115.8333} C_DIS
LIN {X -65.8705,Y -34.176,Z 76,A -157.3295,B 24.9041,C -2.2607,E1 24.8587,E2 -118.2079} C_DIS
LIN {X -64.568,Y -36.5773,Z 76,A -155.2075,B 24.9046,C -2.2554,E1 24.8616,E2 -120.3284} C_DIS
LIN {X -62.9887,Y -39.232,Z 76,A -152.8949,B 24.9052,C -2.2475,E1 24.8649,E2 -122.6341} C_DIS
LIN {X -61.4781,Y -41.5591,Z 76,A -150.759,B 24.9057,C -2.2419,E1 24.8682,E2 -124.7674} C_DIS
LIN {X -59.8111,Y -43.9245,Z 76,A -148.5759,B 24.9063,C -2.2352,E1 24.8717,E2 -126.9452} C_DIS
LIN {X -58.214,Y -46.02,Z 76,A -146.4943,B 24.9066,C -2.2315,E1 24.8753,E2 -129.0279} C_DIS
LIN {X -56.4507,Y -48.1668,Z 76,A -144.1533,B 24.9066,C -2.2314,E1 24.8795,E2 -131.3792} C_DIS
LIN {X -54.3693,Y -50.5065,Z 76,A -141.8122,B 24.9072,C -2.2242,E1 24.8839,E2 -133.7135} C_DIS
LIN {X -52.4734,Y -52.4734,Z 76,A -139.6404,B 24.9074,C -2.2213,E1 24.8882,E2 -135.8876} C_DIS
LIN {X -50.2119,Y -54.6395,Z 76,A -137.3328,B 24.9081,C -2.2137,E1 24.8928,E2 -138.1867} C_DIS
LIN {X -48.1668,Y -56.4507,Z 76,A -135.2144,B 24.9084,C -2.2099,E1 24.8973,E2 -140.3043} C_DIS
LIN {X -45.9691,Y -58.2543,Z 76,A -133.0553,B 24.9088,C -2.205,E1 24.902,E2 -142.46} C_DIS
LIN {X -43.8835,Y -59.8411,Z 76,A -130.9788,B 24.909,C -2.2029,E1 24.9066,E2 -144.5387} C_DIS
LIN {X -41.5591,Y -61.4781,Z 76,A -128.6182,B 24.909,C -2.2035,E1 24.9121,E2 -146.9087} C_DIS
LIN {X -38.9291,Y -63.1779,Z 76,A -126.2808,B 24.9094,C -2.1978,E1 24.9176,E2 -149.24} C_DIS
LIN {X -36.5773,Y -64.568,Z 76,A -124.165,B 24.9096,C -2.195,E1 24.9227,E2 -151.3555} C_DIS
LIN {X -34.176,Y -65.8705,Z 76,A -122.0134,B 24.9098,C -2.1934,E1 24.928,E2 -153.5092} C_DIS
LIN {X -31.3659,Y -67.2525,Z 76,A -119.6938,B 24.9102,C -2.1881,E1 24.9339,E2 -155.8221} C_DIS
LIN {X -28.7668,Y -68.4046,Z 76,A -117.336,B 24.91,C -2.19,E1 24.9399,E2 -158.1899} C_DIS
LIN {X -25.8557,Y -69.5587,Z 76,A -114.9656,B 24.9103,C -2.1865,E1 24.9461,E2 -160.557} C_DIS
LIN {X -22.8976,Y -70.5863,Z 76,A -112.648,B 24.9107,C -2.182,E1 24.9522,E2 -162.8682} C_DIS
LIN {X -20.284,Y -71.3812,Z 76,A -110.5354,B 24.9108,C -2.1806,E1 24.9579,E2 -164.9812} C_DIS
LIN {X -17.5349,Y -72.1058,Z 76,A -108.3824,B 24.911,C -2.1783,E1 24.9637,E2 -167.1317} C_DIS
LIN {X -14.9779,Y -72.68,Z 76,A -106.3119,B 24.911,C -2.1786,E1 24.9694,E2 -169.2056} C_DIS
LIN {X -12.2926,Y -73.182,Z 76,A -104.201,B 24.911,C -2.178,E1 24.9752,E2 -171.3171} C_DIS
LIN {X -9.4804,Y -73.5992,Z 76,A -101.8479,B 24.9107,C -2.1817,E1 24.9817,E2 -173.6808} C_DIS
LIN {X -6.3669,Y -73.935,Z 76,A -99.482,B 24.9108,C -2.1801,E1 24.9883,E2 -176.0443} C_DIS
LIN {X -3.6412,Y -74.1193,Z 76,A -97.4088,B 24.9109,C -2.1793,E1 24.994,E2 -178.116} C_DIS
LIN {X -0.9107,Y -74.2031,Z 76,A -95.3002,B 24.9109,C -2.1796,E1 24.9999,E2 -180.2256} C_DIS
LIN {X -0.9107,Y -74.2031,Z 76,A -95.3002,B 24.9109,C -2.1796,E1 24.9999,E2 -180.2256} C_DIS
Enddeposition()
LIN {X 0.5019,Y -73.2131,Z 76,A -94.7987,B 24.9108,C -2.1813,E1 25.0013,E2 -180.7311} C_DIS
Startdeposition()
$VEL.CP = VEL_PRINT
LIN {X -2.6617,Y -73.1851,Z 76,A -97.8461,B 24.912,C -2.1656,E1 24.9927,E2 -177.6461} C_DIS
LIN {X -5.1665,Y -73.0502,Z 76,A -99.5292,B 24.9114,C -2.1728,E1 24.9881,E2 -175.9796} C_DIS
LIN {X -8.0856,Y -72.7849,Z 76,A -102.5916,B 24.913,C -2.1533,E1 24.9795,E2 -172.8691} C_DIS
LIN {X -12.4679,Y -72.1643,Z 76,A -105.3466,B 24.9115,C -2.1722,E1 24.972,E2 -170.1566} C_DIS
LIN {X -16.5001,Y -71.3493,Z 76,A -108.7531,B 24.9118,C -2.1688,E1 24.9626,E2 -166.738} C_DIS
LIN {X -19.6046,Y -70.5604,Z 76,A -111.269,B 24.9117,C -2.17,E1 24.9558,E2 -164.2212} C_DIS
LIN {X -22.1852,Y -69.7921,Z 76,A -113.4036,B 24.9117,C -2.1709,E1 24.9501,E2 -162.0848} C_DIS
LIN {X -25.0433,Y -68.8172,Z 76,A -115.6722,B 24.9113,C -2.1752,E1 24.9442,E2 -159.8222} C_DIS
LIN {X -28.0369,Y -67.6542,Z 76,A -118.2792,B 24.9113,C -2.1752,E1 24.9374,E2 -157.2096} C_DIS
LIN {X -30.7167,Y -66.4793,Z 76,A -120.5527,B 24.911,C -2.1782,E1 24.9316,E2 -154.9374} C_DIS
LIN {X -32.9566,Y -65.3989,Z 76,A -122.7783,B 24.9114,C -2.1737,E1 24.926,E2 -152.6952} C_DIS
LIN {X -36.2498,Y -63.6318,Z 76,A -125.1238,B 24.9099,C -2.1917,E1 24.9204,E2 -150.386} C_DIS
LIN {X -39.9543,Y -61.3744,Z 76,A -128.9236,B 24.9103,C -2.1868,E1 24.9113,E2 -146.5627} C_DIS
LIN {X -42.5431,Y -59.6075,Z 76,A -131.2384,B 24.9097,C -2.1942,E1 24.906,E2 -144.2575} C_DIS
LIN {X -44.841,Y -57.899,Z 76,A -133.5828,B 24.9096,C -2.1956,E1 24.9008,E2 -141.9079} C_DIS
LIN {X -47.7139,Y -55.5558,Z 76,A -136.4797,B 24.9091,C -2.201,E1 24.8946,E2 -139.0129} C_DIS
LIN {X -49.9367,Y -53.5669,Z 76,A -138.4857,B 24.9081,C -2.2134,E1 24.8905,E2 -137.0284} C_DIS
LIN {X -52.8441,Y -50.7001,Z 76,A -141.7651,B 24.9077,C -2.218,E1 24.884,E2 -133.7462} C_DIS
LIN {X -55.1778,Y -48.1496,Z 76,A -145.1831,B 24.9086,C -2.2073,E1 24.8775,E2 -130.2874} C_DIS
LIN {X -57.9716,Y -44.7468,Z 76,A -148.1085,B 24.9069,C -2.2275,E1 24.8725,E2 -127.3963} C_DIS
LIN {X -60.0389,Y -41.9325,Z 76,A -150.8711,B 24.9064,C -2.2334,E1 24.868,E2 -124.6345} C_DIS
LIN {X -61.5265,Y -39.7177,Z 76,A -152.9897,B 24.906,C -2.238,E1 24.8647,E2 -122.5161} C_DIS
LIN {X -63.0742,Y -37.2106,Z 76,A -155.3892,B 24.9057,C -2.2418,E1 24.8613,E2 -120.1133} C_DIS
LIN {X -64.5478,Y -34.5933,Z 76,A -157.6499,B 24.905,C -2.2501,E1 24.8582,E2 -117.8607} C_DIS
LIN {X -65.9545,Y -31.8275,Z 76,A -160.4753,B 24.9052,C -2.2477,E1 24.8547,E2 -115.0143} C_DIS
LIN {X -67.5637,Y -28.2517,Z 76,A -163.2969,B 24.904,C -2.262,E1 24.8516,E2 -112.2111} C_DIS
LIN {X -68.9836,Y -24.5838,Z 76,A -166.3752,B 24.9033,C -2.2708,E1 24.8486,E2 -109.1367} C_DIS
LIN {X -69.9265,Y -21.7546,Z 76,A -168.7115,B 24.9027,C -2.2777,E1 24.8466,E2 -106.8033} C_DIS
LIN {X -70.7227,Y -19.0074,Z 76,A -171.0087,B 24.9022,C -2.283,E1 24.8449,E2 -104.5056} C_DIS
LIN {X -71.4824,Y -15.9165,Z 76,A -173.4208,B 24.9014,C -2.2923,E1 24.8433,E2 -102.1015} C_DIS
LIN {X -72.0394,Y -13.166,Z 76,A -175.6265,B 24.9008,C -2.2989,E1 24.8421,E2 -99.8984} C_DIS
LIN {X -72.4941,Y -10.3724,Z 76,A -178.0401,B 24.9006,C -2.3013,E1 24.8411,E2 -97.4762} C_DIS
LIN {X -72.9036,Y -6.9342,Z 76,A 179.3653,B 24.8997,C -2.3123,E1 24.8404,E2 -94.8924} C_DIS
LIN {X -73.1348,Y -3.7872,Z 76,A 176.8407,B 24.8991,C -2.3188,E1 24.8399,E2 -92.3682} C_DIS
LIN {X -73.2303,Y -0.6015,Z 76,A 174.3888,B 24.8983,C -2.3277,E1 24.8398,E2 -89.9226} C_DIS
LIN {X -73.2047,Y 2.0241,Z 76,A 172.2947,B 24.8978,C -2.3333,E1 24.8398,E2 -87.8294} C_DIS
LIN {X -73.0527,Y 5.1299,Z 76,A 169.8432,B 24.8972,C -2.3406,E1 24.8403,E2 -85.3806} C_DIS
LIN {X -72.7824,Y 8.1159,Z 76,A 167.4579,B 24.8966,C -2.3472,E1 24.841,E2 -82.9966} C_DIS
LIN {X -72.3886,Y 11.0846,Z 76,A 165.4307,B 24.8953,C -2.3617,E1 24.8417,E2 -80.9919} C_DIS
LIN {X -72.0285,Y 13.2266,Z 76,A 163.2213,B 24.8959,C -2.3556,E1 24.8428,E2 -78.755} C_DIS
LIN {X -71.3243,Y 16.6082,Z 76,A 160.714,B 24.8947,C -2.3685,E1 24.8443,E2 -76.2637} C_DIS
LIN {X -70.585,Y 19.5169,Z 76,A 158.2318,B 24.8944,C -2.3728,E1 24.8461,E2 -73.7773} C_DIS
LIN {X -69.5675,Y 22.8792,Z 76,A 155.5191,B 24.8935,C -2.382,E1 24.8484,E2 -71.0712} C_DIS
LIN {X -68.5672,Y 25.7211,Z 76,A 153.245,B 24.8927,C -2.3911,E1 24.8505,E2 -68.8058} C_DIS
LIN {X -67.7189,Y 27.8774,Z 76,A 151.4541,B 24.8922,C -2.3971,E1 24.8524,E2 -67.0192} C_DIS
LIN {X -66.5982,Y 30.4571,Z 76,A 148.6717,B 24.8928,C -2.3906,E1 24.8556,E2 -64.2061} C_DIS
LIN {X -64.2448,Y 35.1518,Z 76,A 144.7093,B 24.8914,C -2.4058,E1 24.8607,E2 -60.2589} C_DIS
LIN {X -62.2781,Y 38.5294,Z 76,A 141.8688,B 24.8902,C -2.4193,E1 24.8648,E2 -57.4359} C_DIS
LIN {X -60.389,Y 41.4285,Z 76,A 139.1188,B 24.8896,C -2.4258,E1 24.8691,E2 -54.6876} C_DIS
LIN {X -58.5698,Y 43.9608,Z 76,A 136.8645,B 24.8886,C -2.4365,E1 24.8728,E2 -52.4482} C_DIS
LIN {X -56.7782,Y 46.252,Z 76,A 134.5052,B 24.8882,C -2.4405,E1 24.8769,E2 -50.0874} C_DIS
LIN {X -54.8431,Y 48.5322,Z 76,A 132.1027,B 24.8878,C -2.445,E1 24.8813,E2 -47.6846} C_DIS
LIN {X -52.8553,Y 50.6885,Z 76,A 130.0223,B 24.8868,C -2.4555,E1 24.8852,E2 -45.6202} C_DIS
LIN {X -51.2923,Y 52.2698,Z 76,A 128.036,B 24.887,C -2.454,E1 24.8891,E2 -43.6218} C_DIS
LIN {X -49.0885,Y 54.3451,Z 76,A 125.6666,B 24.8865,C -2.4594,E1 24.894,E2 -41.2557} C_DIS
LIN {X -46.8074,Y 56.3209,Z 76,A 123.3149,B 24.886,C -2.4648,E1 24.899,E2 -38.9079} C_DIS
LIN {X -44.6879,Y 58.0169,Z 76,A 121.4078,B 24.8851,C -2.4744,E1 24.9031,E2 -37.0165} C_DIS
LIN {X -42.8463,Y 59.3912,Z 76,A 119.3564,B 24.8853,C -2.4721,E1 24.9078,E2 -34.9524} C_DIS
LIN {X -40.5073,Y 61.0097,Z 76,A 117.1664,B 24.8848,C -2.4772,E1 24.9128,E2 -32.7673} C_DIS
LIN {X -38.125,Y 62.5257,Z 76,A 114.9742,B 24.8844,C -2.4817,E1 24.918,E2 -30.5789} C_DIS
LIN {X -35.3588,Y 64.1318,Z 76,A 112.4951,B 24.8839,C -2.4866,E1 24.924,E2 -28.1041} C_DIS
LIN {X -33.6596,Y 65.0395,Z 76,A 110.4429,B 24.8849,C -2.4761,E1 24.9292,E2 -26.0214} C_DIS
LIN {X -29.8168,Y 66.8881,Z 76,A 107.5077,B 24.8836,C -2.4907,E1 24.9366,E2 -23.1136} C_DIS
LIN {X -27.3002,Y 67.9543,Z 76,A 105.6472,B 24.8827,C -2.5004,E1 24.9413,E2 -21.272} C_DIS
LIN {X -23.6278,Y 69.3161,Z 76,A 102.3457,B 24.8828,C -2.4985,E1 24.95,E2 -17.9593} C_DIS
LIN {X -20.7537,Y 70.2301,Z 76,A 99.9446,B 24.8827,C -2.5001,E1 24.9564,E2 -15.558} C_DIS
LIN {X -17.779,Y 71.0424,Z 76,A 97.5895,B 24.8823,C -2.5039,E1 24.9628,E2 -13.2084} C_DIS
LIN {X -14.001,Y 71.8816,Z 76,A 94.9273,B 24.8812,C -2.5156,E1 24.97,E2 -10.5707} C_DIS
LIN {X -10.6165,Y 72.4594,Z 76,A 91.1727,B 24.8835,C -2.491,E1 24.9805,E2 -6.7542} C_DIS
LIN {X -4.7161,Y 73.0807,Z 76,A 86.7282,B 24.8829,C -2.4981,E1 24.9928,E2 -2.3244} C_DIS
LIN {X -0.8518,Y 73.2283,Z 76,A 83.8705,B 24.8824,C -2.503,E1 25.0008,E2 0.5216} C_DIS
LIN {X 3.3113,Y 73.1576,Z 76,A 81.1076,B 24.8812,C -2.516,E1 25.0084,E2 3.2533} C_DIS
LIN {X 5.039,Y 73.0588,Z 76,A 78.8921,B 24.8832,C -2.494,E1 25.0147,E2 5.5199} C_DIS
LIN {X 8.2471,Y 72.767,Z 76,A 76.5039,B 24.883,C -2.497,E1 25.0213,E2 7.8994} C_DIS
LIN {X 13.4364,Y 71.9904,Z 76,A 72.8531,B 24.882,C -2.5073,E1 25.0313,E2 11.5219} C_DIS
LIN {X 16.4497,Y 71.3609,Z 76,A 70.4911,B 24.882,C -2.5073,E1 25.0377,E2 13.8807} C_DIS
LIN {X 19.4667,Y 70.5986,Z 76,A 67.9816,B 24.8823,C -2.5039,E1 25.0445,E2 16.3945} C_DIS
LIN {X 22.3707,Y 69.7321,Z 76,A 65.7362,B 24.8822,C -2.5054,E1 25.0505,E2 18.6323} C_DIS
LIN {X 25.2463,Y 68.7432,Z 76,A 63.2559,B 24.8826,C -2.5007,E1 25.057,E2 21.1189} C_DIS
LIN {X 28.1666,Y 67.5996,Z 76,A 60.9626,B 24.8825,C -2.5024,E1 25.0629,E2 23.4026} C_DIS
LIN {X 31.5388,Y 66.0932,Z 76,A 58.0208,B 24.8829,C -2.4978,E1 25.0704,E2 26.3481} C_DIS
LIN {X 34.1712,Y 64.7712,Z 76,A 55.9694,B 24.8825,C -2.5017,E1 25.0755,E2 28.3847} C_DIS
LIN {X 37.2833,Y 63.0312,Z 76,A 52.8473,B 24.8837,C -2.4888,E1 25.0831,E2 31.5281} C_DIS
LIN {X 40.0318,Y 61.3233,Z 76,A 50.3777,B 24.8839,C -2.4866,E1 25.0889,E2 33.9949} C_DIS
LIN {X 42.4946,Y 59.6421,Z 76,A 48.0777,B 24.8842,C -2.4836,E1 25.0942,E2 36.2939} C_DIS
LIN {X 44.8516,Y 57.8908,Z 76,A 45.9046,B 24.8842,C -2.483,E1 25.099,E2 38.4606} C_DIS
LIN {X 47.4716,Y 55.7622,Z 76,A 42.9581,B 24.8855,C -2.4697,E1 25.1054,E2 41.4274} C_DIS
LIN {X 50.8135,Y 52.7348,Z 76,A 39.6327,B 24.8857,C -2.4682,E1 25.1122,E2 44.7428} C_DIS
LIN {X 52.9053,Y 50.6367,Z 76,A 37.4958,B 24.8857,C -2.4682,E1 25.1163,E2 46.8704} C_DIS
LIN {X 54.7378,Y 48.6499,Z 76,A 34.9379,B 24.8872,C -2.4512,E1 25.1212,E2 49.4572} C_DIS
LIN {X 56.6559,Y 46.4024,Z 76,A 32.4227,B 24.8882,C -2.4402,E1 25.1257,E2 51.9868} C_DIS
LIN {X 60.0308,Y 41.9442,Z 76,A 28.5421,B 24.888,C -2.4434,E1 25.132,E2 55.8412} C_DIS
LIN {X 61.7562,Y 39.3598,Z 76,A 26.1372,B 24.8885,C -2.438,E1 25.1357,E2 58.247} C_DIS
LIN {X 63.7741,Y 35.9994,Z 76,A 23.0605,B 24.8892,C -2.4296,E1 25.1401,E2 61.3276} C_DIS
LIN {X 65.3216,Y 33.1077,Z 76,A 20.6076,B 24.8896,C -2.4258,E1 25.1432,E2 63.7765} C_DIS
LIN {X 66.5436,Y 30.5786,Z 76,A 18.6289,B 24.8896,C -2.426,E1 25.1456,E2 65.7441} C_DIS
LIN {X 67.595,Y 28.1776,Z 76,A 16.3449,B 24.8907,C -2.4135,E1 25.1481,E2 68.0451} C_DIS
LIN {X 68.6529,Y 25.4939,Z 76,A 14.0495,B 24.8914,C -2.4058,E1 25.1504,E2 70.3459} C_DIS
LIN {X 69.6529,Y 22.6153,Z 76,A 11.7776,B 24.8917,C -2.4021,E1 25.1524,E2 72.6138} C_DIS
LIN {X 70.6202,Y 19.3868,Z 76,A 9.0798,B 24.8926,C -2.3924,E1 25.1545,E2 75.319} C_DIS
LIN {X 71.3645,Y 16.4342,Z 76,A 6.9909,B 24.8925,C -2.3937,E1 25.1559,E2 77.3929} C_DIS
LIN {X 72.0708,Y 12.9906,Z 76,A 3.6575,B 24.8947,C -2.3684,E1 25.1577,E2 80.7665} C_DIS
LIN {X 72.6851,Y 8.946,Z 76,A 0.7497,B 24.8949,C -2.3668,E1 25.1588,E2 83.6608} C_DIS
LIN {X 72.9842,Y 6.026,Z 76,A -1.7,B 24.8959,C -2.3552,E1 25.1594,E2 86.1235} C_DIS
LIN {X 73.2274,Y 0.9392,Z 76,A -5.2689,B 24.8959,C -2.3546,E1 25.1598,E2 89.6725} C_DIS
LIN {X 73.1593,Y -3.2714,Z 76,A -8.4906,B 24.8967,C -2.3463,E1 25.1596,E2 92.8948} C_DIS
LIN {X 73.0078,Y -5.731,Z 76,A -10.526,B 24.8975,C -2.337,E1 25.1592,E2 94.94} C_DIS
LIN {X 72.5588,Y -9.9172,Z 76,A -13.9527,B 24.8988,C -2.3227,E1 25.1581,E2 98.3803} C_DIS
LIN {X 72.0078,Y -13.3414,Z 76,A -16.6093,B 24.8994,C -2.3158,E1 25.1568,E2 101.0376} C_DIS
LIN {X 71.3205,Y -16.6249,Z 76,A -19.6473,B 24.9011,C -2.2956,E1 25.1549,E2 104.1057} C_DIS
LIN {X 70.3197,Y -20.4515,Z 76,A -22.1654,B 24.9005,C -2.3026,E1 25.1531,E2 106.5928} C_DIS
LIN {X 69.2181,Y -23.9154,Z 76,A -25.1369,B 24.9016,C -2.2901,E1 25.1505,E2 109.577} C_DIS
LIN {X 68.0278,Y -27.117,Z 76,A -27.7938,B 24.9023,C -2.2824,E1 25.1478,E2 112.2373} C_DIS
LIN {X 66.8947,Y -29.8021,Z 76,A -30.0495,B 24.9028,C -2.2763,E1 25.1453,E2 114.4951} C_DIS
LIN {X 65.433,Y -32.8887,Z 76,A -32.7389,B 24.9035,C -2.2679,E1 25.142,E2 117.19} C_DIS
LIN {X 63.9381,Y -35.7056,Z 76,A -35.1618,B 24.9039,C -2.2627,E1 25.1388,E2 119.6123} C_DIS
LIN {X 62.3375,Y -38.4342,Z 76,A -37.6414,B 24.9046,C -2.2556,E1 25.1352,E2 122.0961} C_DIS
LIN {X 60.6462,Y -41.0489,Z 76,A -39.7408,B 24.9043,C -2.2585,E1 25.132,E2 124.1781} C_DIS
LIN {X 58.7431,Y -43.7301,Z 76,A -42.3499,B 24.905,C -2.2505,E1 25.1277,E2 126.7935} C_DIS
LIN {X 56.7049,Y -46.3424,Z 76,A -45.482,B 24.9069,C -2.2283,E1 25.1222,E2 129.9635} C_DIS
LIN {X 54.6418,Y -48.7572,Z 76,A -48.6239,B 24.9089,C -2.2035,E1 25.1163,E2 133.15} C_DIS
LIN {X 51.7075,Y -51.8597,Z 76,A -50.9776,B 24.9073,C -2.2231,E1 25.1118,E2 135.4472} C_DIS
LIN {X 50.1708,Y -53.3466,Z 76,A -53.1769,B 24.9088,C -2.2044,E1 25.1072,E2 137.6817} C_DIS
LIN {X 46.0445,Y -56.9463,Z 76,A -57.2313,B 24.9091,C -2.2014,E1 25.0986,E2 141.7277} C_DIS
LIN {X 43.4503,Y -58.95,Z 76,A -60.3091,B 24.9107,C -2.1818,E1 25.0916,E2 144.8407} C_DIS
LIN {X 40.2439,Y -61.1834,Z 76,A -61.9618,B 24.908,C -2.2149,E1 25.088,E2 146.4097} C_DIS
LIN {X 36.2848,Y -63.6116,Z 76,A -66.0896,B 24.9097,C -2.1943,E1 25.0781,E2 150.5731} C_DIS
LIN {X 33.6537,Y -65.0426,Z 76,A -68.497,B 24.9102,C -2.1886,E1 25.0721,E2 152.9874} C_DIS
LIN {X 30.6163,Y -66.5261,Z 76,A -71.0168,B 24.9102,C -2.1879,E1 25.0657,E2 155.5023} C_DIS
LIN {X 27.9048,Y -67.7082,Z 76,A -73.427,B 24.9107,C -2.1819,E1 25.0595,E2 157.921} C_DIS
LIN {X 24.7509,Y -68.9239,Z 76,A -76.0576,B 24.911,C -2.1788,E1 25.0526,E2 160.5535} C_DIS
LIN {X 22.0493,Y -69.8351,Z 76,A -78.5827,B 24.9118,C -2.1682,E1 25.0459,E2 163.0989} C_DIS
LIN {X 18.3913,Y -70.8856,Z 76,A -81.0461,B 24.911,C -2.1789,E1 25.0393,E2 165.533} C_DIS
LIN {X 14.733,Y -71.735,Z 76,A -84.08,B 24.9114,C -2.1736,E1 25.031,E2 168.5754} C_DIS
LIN {X 11.7619,Y -72.2823,Z 76,A -86.5133,B 24.9117,C -2.1699,E1 25.0243,E2 171.0148} C_DIS
LIN {X 8.748,Y -72.7083,Z 76,A -88.9051,B 24.9118,C -2.1681,E1 25.0177,E2 173.4089} C_DIS
LIN {X 4.3127,Y -73.1057,Z 76,A -92.3359,B 24.9118,C -2.1678,E1 25.0081,E2 176.8385} C_DIS
LIN {X 2.0792,Y -73.203,Z 76,A -94.7258,B 24.9133,C -2.1506,E1 25.0014,E2 179.2689} C_DIS
LIN {X 2.0792,Y -73.203,Z 76,A -94.7258,B 24.9133,C -2.1506,E1 25.0014,E2 179.2689} C_DIS
Enddeposition()
LIN {X 0.4881,Y -72.2305,Z 76,A -94.4255,B 24.9086,C -2.208,E1 25.0026,E2 178.8324} C_DIS
Startdeposition()
$VEL.CP = VEL_PRINT
LIN {X 4.5391,Y -72.1155,Z 76,A -90.5341,B 24.907,C -2.2267,E1 25.0135,E2 174.8978} C_DIS
LIN {X 10.126,Y -71.5444,Z 76,A -86.6959,B 24.9081,C -2.2129,E1 25.0241,E2 171.0953} C_DIS
LIN {X 14.1538,Y -70.8586,Z 76,A -82.9566,B 24.9068,C -2.2289,E1 25.0344,E2 167.3221} C_DIS
LIN {X 18.3643,Y -69.8859,Z 76,A -79.9228,B 24.9074,C -2.2216,E1 25.0426,E2 164.3101} C_DIS
LIN {X 23.9455,Y -68.1744,Z 76,A -75.3518,B 24.9071,C -2.2255,E1 25.0548,E2 159.7384} C_DIS
LIN {X 26.7753,Y -67.1146,Z 76,A -72.8539,B 24.9066,C -2.2315,E1 25.0613,E2 157.2316} C_DIS
LIN {X 29.6677,Y -65.886,Z 76,A -70.6055,B 24.9068,C -2.2285,E1 25.067,E2 154.9958} C_DIS
LIN {X 33.1314,Y -64.2146,Z 76,A -67.2993,B 24.9058,C -2.2405,E1 25.0753,E2 151.67} C_DIS
LIN {X 36.1339,Y -62.5739,Z 76,A -63.9899,B 24.904,C -2.2621,E1 25.0835,E2 148.3196} C_DIS
LIN {X 39.0663,Y -60.7862,Z 76,A -62.1617,B 24.9057,C -2.242,E1 25.0877,E2 146.5446} C_DIS
LIN {X 42.0852,Y -58.7366,Z 76,A -59.2606,B 24.9052,C -2.248,E1 25.0943,E2 143.6393} C_DIS
LIN {X 43.8742,Y -57.4128,Z 76,A -57.0546,B 24.9038,C -2.2642,E1 25.0993,E2 141.4031} C_DIS
LIN {X 47.1501,Y -54.7553,Z 76,A -53.7778,B 24.9034,C -2.2696,E1 25.1063,E2 138.126} C_DIS
LIN {X 50.5327,Y -51.6493,Z 76,A -50.5107,B 24.9035,C -2.2675,E1 25.1129,E2 134.8774} C_DIS
LIN {X 53.0944,Y -49.0119,Z 76,A -47.2892,B 24.9022,C -2.2834,E1 25.1192,E2 131.6322} C_DIS
LIN {X 55.7207,Y -46.0042,Z 76,A -44.0807,B 24.9014,C -2.2928,E1 25.125,E2 128.4162} C_DIS
LIN {X 57.7576,Y -43.4189,Z 76,A -41.8175,B 24.9016,C -2.2897,E1 25.1288,E2 126.171} C_DIS
LIN {X 59.8959,Y -40.4181,Z 76,A -38.7999,B 24.9007,C -2.3004,E1 25.1336,E2 123.1428} C_DIS
LIN {X 61.6445,Y -37.6979,Z 76,A -36.3788,B 24.9004,C -2.3035,E1 25.1372,E2 120.7267} C_DIS
LIN {X 63.3078,Y -34.8333,Z 76,A -33.2235,B 24.8985,C -2.3264,E1 25.1416,E2 117.5337} C_DIS
LIN {X 65.2951,Y -30.9488,Z 76,A -30.23,B 24.8987,C -2.323,E1 25.1452,E2 114.5642} C_DIS
LIN {X 66.564,Y -28.1135,Z 76,A -27.8641,B 24.8983,C -2.3276,E1 25.1479,E2 112.2004} C_DIS
LIN {X 67.7027,Y -25.2509,Z 76,A -24.8458,B 24.8962,C -2.3518,E1 25.1509,E2 109.1417} C_DIS
LIN {X 69.173,Y -20.8891,Z 76,A -21.9376,B 24.8971,C -2.3414,E1 25.1533,E2 106.2745} C_DIS
LIN {X 69.8881,Y -18.3534,Z 76,A -19.7164,B 24.8962,C -2.3518,E1 25.155,E2 104.0416} C_DIS
LIN {X 70.5243,Y -15.7346,Z 76,A -17.4686,B 24.8953,C -2.3617,E1 25.1564,E2 101.7834} C_DIS
LIN {X 71.2998,Y -11.7262,Z 76,A -14.7826,B 24.8959,C -2.3559,E1 25.1577,E2 99.1268} C_DIS
LIN {X 71.7648,Y -8.4226,Z 76,A -11.1613,B 24.8926,C -2.3928,E1 25.1591,E2 95.4397} C_DIS
LIN {X 72.1187,Y -4.4824,Z 76,A -8.331,B 24.8925,C -2.3938,E1 25.1596,E2 92.6239} C_DIS
LIN {X 72.2583,Y 0.0149,Z 76,A -5.3545,B 24.893,C -2.3879,E1 25.1598,E2 89.6792} C_DIS
LIN {X 72.1871,Y 3.1787,Z 76,A -2.4162,B 24.8912,C -2.4083,E1 25.1595,E2 86.71} C_DIS
LIN {X 71.8868,Y 7.3051,Z 76,A 1.0824,B 24.8896,C -2.425,E1 25.1586,E2 83.1927} C_DIS
LIN {X 71.1169,Y 12.7875,Z 76,A 5.5892,B 24.8881,C -2.442,E1 25.1566,E2 78.6723} C_DIS
LIN {X 70.1532,Y 17.3117,Z 76,A 8.6088,B 24.8888,C -2.4343,E1 25.1548,E2 75.6885} C_DIS
LIN {X 69.4732,Y 19.8653,Z 76,A 10.949,B 24.8876,C -2.4477,E1 25.153,E2 73.33} C_DIS
LIN {X 68.4113,Y 23.2608,Z 76,A 13.5351,B 24.8874,C -2.4492,E1 25.1508,E2 70.755} C_DIS
LIN {X 67.4291,Y 25.9735,Z 76,A 15.5996,B 24.8874,C -2.4494,E1 25.1488,E2 68.7015} C_DIS
LIN {X 66.4737,Y 28.3278,Z 76,A 18.0513,B 24.8857,C -2.4677,E1 25.1461,E2 66.22} C_DIS
LIN {X 64.505,Y 32.5633,Z 76,A 21.563,B 24.8853,C -2.4724,E1 25.1419,E2 62.716} C_DIS
LIN {X 61.5728,Y 37.8159,Z 76,A 26.2675,B 24.8843,C -2.4832,E1 25.1354,E2 58.0105} C_DIS
LIN {X 60.0057,Y 40.256,Z 76,A 28.9024,B 24.8828,C -2.4985,E1 25.1313,E2 55.3523} C_DIS
LIN {X 57.7523,Y 43.4259,Z 76,A 31.603,B 24.8831,C -2.4952,E1 25.1268,E2 52.6727} C_DIS
LIN {X 55.3101,Y 46.4983,Z 76,A 34.4788,B 24.8831,C -2.4958,E1 25.1218,E2 49.8088} C_DIS
LIN {X 52.7215,Y 49.4124,Z 76,A 38.4302,B 24.8801,C -2.5268,E1 25.1143,E2 45.8015} C_DIS
LIN {X 50.4402,Y 51.7406,Z 76,A 41.1196,B 24.8794,C -2.5351,E1 25.1089,E2 43.1037} C_DIS
LIN {X 47.8883,Y 54.1097,Z 76,A 43.6886,B 24.8794,C -2.5351,E1 25.1035,E2 40.5449} C_DIS
LIN {X 44.4264,Y 56.9877,Z 76,A 46.7914,B 24.88,C -2.5287,E1 25.0968,E2 37.469} C_DIS
LIN {X 41.7874,Y 58.9491,Z 76,A 49.2856,B 24.8798,C -2.53,E1 25.0912,E2 34.9805} C_DIS
LIN {X 39.3761,Y 60.5873,Z 76,A 51.5901,B 24.8795,C -2.5334,E1 25.0858,E2 32.6754} C_DIS
LIN {X 36.9773,Y 62.0796,Z 76,A 54.3163,B 24.8779,C -2.55,E1 25.0792,E2 29.9184} C_DIS
LIN {X 31.8008,Y 64.8841,Z 76,A 59.146,B 24.8769,C -2.5603,E1 25.0672,E2 25.0776} C_DIS
LIN {X 28.7964,Y 66.2715,Z 76,A 61.1841,B 24.8782,C -2.5474,E1 25.0621,E2 23.0751} C_DIS
LIN {X 25.6447,Y 67.5536,Z 76,A 63.7886,B 24.8782,C -2.5475,E1 25.0553,E2 20.4761} C_DIS
LIN {X 22.6192,Y 68.627,Z 76,A 66.311,B 24.878,C -2.549,E1 25.0487,E2 17.9551} C_DIS
LIN {X 19.5606,Y 69.5596,Z 76,A 68.9025,B 24.8777,C -2.5523,E1 25.0417,E2 15.3602} C_DIS
LIN {X 16.3705,Y 70.3786,Z 76,A 71.483,B 24.8777,C -2.553,E1 25.0347,E2 12.7819} C_DIS
LIN {X 13.2897,Y 71.0258,Z 76,A 74.2471,B 24.8769,C -2.561,E1 25.0271,E2 10.0021} C_DIS
LIN {X 8.8654,Y 71.7115,Z 76,A 77.5264,B 24.8775,C -2.5549,E1 25.0181,E2 6.7402} C_DIS
LIN {X 5.2382,Y 72.0677,Z 76,A 80.4355,B 24.8774,C -2.5556,E1 25.01,E2 3.831} C_DIS
LIN {X 2.0435,Y 72.2287,Z 76,A 82.9965,B 24.8774,C -2.556,E1 25.0028,E2 1.2696} C_DIS
LIN {X -1.2292,Y 72.247,Z 76,A 85.6511,B 24.8773,C -2.557,E1 24.9954,E2 -1.3872} C_DIS
LIN {X -4.8437,Y 72.0949,Z 76,A 88.5273,B 24.8773,C -2.5561,E1 24.9874,E2 -4.2622} C_DIS
LIN {X -7.8032,Y 71.8354,Z 76,A 91.1248,B 24.8769,C -2.561,E1 24.9802,E2 -6.8727} C_DIS
LIN {X -12.7158,Y 71.1298,Z 76,A 94.5673,B 24.8783,C -2.546,E1 24.9708,E2 -10.2826} C_DIS
LIN {X -15.2754,Y 70.6244,Z 76,A 96.8144,B 24.8781,C -2.5486,E1 24.9646,E2 -12.5387} C_DIS
LIN {X -18.4183,Y 69.8719,Z 76,A 99.3986,B 24.8782,C -2.5467,E1 24.9576,E2 -15.122} C_DIS
LIN {X -21.4313,Y 69.006,Z 76,A 101.6175,B 24.8791,C -2.5375,E1 24.9517,E2 -17.3227} C_DIS
LIN {X -24.3703,Y 68.0246,Z 76,A 104.1783,B 24.8791,C -2.537,E1 24.9449,E2 -19.8872} C_DIS
LIN {X -26.4296,Y 67.2504,Z 76,A 106.7948,B 24.8774,C -2.5559,E1 24.938,E2 -22.5544} C_DIS
LIN {X -29.6759,Y 65.8823,Z 76,A 108.6492,B 24.8799,C -2.5291,E1 24.9334,E2 -24.3494} C_DIS
LIN {X -31.6038,Y 64.9802,Z 76,A 110.9648,B 24.8787,C -2.5415,E1 24.9275,E2 -26.7006} C_DIS
LIN {X -35.6855,Y 62.8316,Z 76,A 114.2349,B 24.8802,C -2.5261,E1 24.9196,E2 -29.9432} C_DIS
LIN {X -38.3392,Y 61.2474,Z 76,A 116.6568,B 24.8807,C -2.5209,E1 24.9138,E2 -32.3604} C_DIS
LIN {X -40.8083,Y 59.6318,Z 76,A 118.8339,B 24.8815,C -2.5126,E1 24.9088,E2 -34.5247} C_DIS
LIN {X -43.4883,Y 57.7054,Z 76,A 121.8369,B 24.8811,C -2.5163,E1 24.902,E2 -37.5473} C_DIS
LIN {X -46.3338,Y 55.4468,Z 76,A 124.5333,B 24.8821,C -2.5058,E1 24.8962,E2 -40.2288} C_DIS
LIN {X -48.5909,Y 53.4807,Z 76,A 126.9322,B 24.8826,C -2.501,E1 24.8912,E2 -42.6259} C_DIS
LIN {X -50.3514,Y 51.8261,Z 76,A 128.9547,B 24.8828,C -2.4991,E1 24.8871,E2 -44.652} C_DIS
LIN {X -53.0611,Y 49.0482,Z 76,A 131.9249,B 24.8837,C -2.4891,E1 24.8814,E2 -47.6113} C_DIS
LIN {X -55.0296,Y 46.8281,Z 76,A 134.2575,B 24.8843,C -2.4827,E1 24.8771,E2 -49.9392} C_DIS
LIN {X -56.8773,Y 44.5667,Z 76,A 136.8155,B 24.8843,C -2.4823,E1 24.8727,E2 -52.5081} C_DIS
LIN {X -59.7638,Y 40.6133,Z 76,A 140.5678,B 24.8856,C -2.4688,E1 24.8666,E2 -56.2466} C_DIS
LIN {X -61.4661,Y 37.989,Z 76,A 143.0496,B 24.8862,C -2.4619,E1 24.8629,E2 -58.7246} C_DIS
LIN {X -64.1736,Y 33.2118,Z 76,A 147.147,B 24.8879,C -2.4436,E1 24.8574,E2 -62.7998} C_DIS
LIN {X -66.2673,Y 28.8059,Z 76,A 151.1491,B 24.8887,C -2.4352,E1 24.8527,E2 -66.8035} C_DIS
LIN {X -67.4554,Y 25.9039,Z 76,A 153.8424,B 24.889,C -2.4323,E1 24.8499,E2 -69.505} C_DIS
LIN {X -68.5351,Y 22.8937,Z 76,A 156.4259,B 24.8896,C -2.4256,E1 24.8475,E2 -72.0873} C_DIS
LIN {X -69.4771,Y 19.8518,Z 76,A 158.9423,B 24.8903,C -2.4176,E1 24.8455,E2 -74.5991} C_DIS
LIN {X -70.3063,Y 16.6836,Z 76,A 161.2961,B 24.8915,C -2.404,E1 24.8439,E2 -76.9342} C_DIS
LIN {X -70.9483,Y 13.6919,Z 76,A 163.559,B 24.8926,C -2.3928,E1 24.8426,E2 -79.1835} C_DIS
LIN {X -71.4602,Y 10.7088,Z 76,A 166.428,B 24.8923,C -2.3957,E1 24.8413,E2 -82.0765} C_DIS
LIN {X -71.836,Y 7.7973,Z 76,A 168.7328,B 24.893,C -2.3878,E1 24.8405,E2 -84.3762} C_DIS
LIN {X -72.0993,Y 4.7788,Z 76,A 170.9275,B 24.8941,C -2.3755,E1 24.8401,E2 -86.5548} C_DIS
LIN {X -72.2231,Y 2.2271,Z 76,A 173.2653,B 24.8941,C -2.3761,E1 24.8398,E2 -88.9079} C_DIS
LIN {X -72.2497,Y -1.082,Z 76,A 175.8572,B 24.8949,C -2.367,E1 24.8398,E2 -91.4939} C_DIS
LIN {X -72.126,Y -4.3725,Z 76,A 178.4532,B 24.8956,C -2.3584,E1 24.8402,E2 -94.085} C_DIS
LIN {X -71.9762,Y -6.3738,Z 76,A -179.7834,B 24.8957,C -2.3573,E1 24.8406,E2 -95.8563} C_DIS
LIN {X -71.3722,Y -11.278,Z 76,A -175.9362,B 24.8969,C -2.3435,E1 24.8421,E2 -99.6935} C_DIS
LIN {X -70.7907,Y -14.485,Z 76,A -173.5661,B 24.8981,C -2.3307,E1 24.8433,E2 -102.0471} C_DIS
LIN {X -70.0593,Y -17.6895,Z 76,A -169.9616,B 24.8968,C -2.3456,E1 24.8457,E2 -105.7081} C_DIS
LIN {X -69.0949,Y -21.1448,Z 76,A -167.8836,B 24.8991,C -2.3196,E1 24.8473,E2 -107.736} C_DIS
LIN {X -68.267,Y -23.6817,Z 76,A -165.2414,B 24.8985,C -2.3254,E1 24.8498,E2 -110.4072} C_DIS
LIN {X -66.8012,Y -27.5471,Z 76,A -161.5338,B 24.8985,C -2.326,E1 24.8537,E2 -114.1369} C_DIS
LIN {X -65.2035,Y -31.1395,Z 76,A -159.5272,B 24.9015,C -2.2916,E1 24.856,E2 -116.0724} C_DIS
LIN {X -63.3138,Y -34.8235,Z 76,A -155.9422,B 24.9016,C -2.2897,E1 24.8607,E2 -119.6717} C_DIS
LIN {X -61.7286,Y -37.5595,Z 76,A -153.5132,B 24.9024,C -2.2813,E1 24.8641,E2 -122.0933} C_DIS
LIN {X -60.1403,Y -40.0548,Z 76,A -150.268,B 24.9011,C -2.2965,E1 24.8692,E2 -125.391} C_DIS
LIN {X -57.9527,Y -43.1591,Z 76,A -148.1437,B 24.9035,C -2.2683,E1 24.8726,E2 -127.4583} C_DIS
LIN {X -55.9151,Y -45.7685,Z 76,A -144.485,B 24.9019,C -2.2866,E1 24.8792,E2 -131.1778} C_DIS
LIN {X -53.2405,Y -48.8527,Z 76,A -142.274,B 24.9046,C -2.2551,E1 24.8832,E2 -133.3233} C_DIS
LIN {X -51.6272,Y -50.5556,Z 76,A -139.9416,B 24.904,C -2.2623,E1 24.8878,E2 -135.6832} C_DIS
LIN {X -48.7095,Y -53.3719,Z 76,A -137.3553,B 24.9058,C -2.2409,E1 24.8929,E2 -138.2288} C_DIS
LIN {X -46.7573,Y -55.09,Z 76,A -134.4409,B 24.9044,C -2.2574,E1 24.8992,E2 -141.1941} C_DIS
LIN {X -43.0472,Y -58.0366,Z 76,A -131.172,B 24.906,C -2.239,E1 24.9064,E2 -144.4309} C_DIS
LIN {X -40.1948,Y -60.0471,Z 76,A -128.7562,B 24.907,C -2.226,E1 24.9119,E2 -146.8239} C_DIS
LIN {X -37.5622,Y -61.727,Z 76,A -125.6593,B 24.9061,C -2.2375,E1 24.9193,E2 -149.9579} C_DIS
LIN {X -34.3717,Y -63.5589,Z 76,A -123.3799,B 24.9077,C -2.2179,E1 24.9248,E2 -152.1973} C_DIS
LIN {X -31.7241,Y -64.9221,Z 76,A -120.6128,B 24.9071,C -2.225,E1 24.9317,E2 -154.9886} C_DIS
LIN {X -28.8728,Y -66.2382,Z 76,A -118.1697,B 24.9075,C -2.2211,E1 24.938,E2 -157.4284} C_DIS
LIN {X -25.8702,Y -67.4682,Z 76,A -115.6157,B 24.9077,C -2.2182,E1 24.9446,E2 -159.9809} C_DIS
LIN {X -22.3238,Y -68.7225,Z 76,A -112.6298,B 24.9079,C -2.2158,E1 24.9525,E2 -162.967} C_DIS
LIN {X -19.4982,Y -69.5773,Z 76,A -110.2558,B 24.9079,C -2.2151,E1 24.9588,E2 -165.3431} C_DIS
LIN {X -16.3516,Y -70.383,Z 76,A -107.3007,B 24.9073,C -2.2235,E1 24.9669,E2 -168.3222} C_DIS
LIN {X -11.3709,Y -71.3579,Z 76,A -104.0083,B 24.9089,C -2.2033,E1 24.9759,E2 -171.57} C_DIS
LIN {X -8.3638,Y -71.7717,Z 76,A -101.113,B 24.9079,C -2.2154,E1 24.984,E2 -174.4964} C_DIS
LIN {X -4.5126,Y -72.1162,Z 76,A -97.933,B 24.9077,C -2.2184,E1 24.9928,E2 -177.6846} C_DIS
LIN {X -0.9945,Y -72.2513,Z 76,A -94.4922,B 24.9062,C -2.2361,E1 25.0026,E2 -181.1676} C_DIS
LIN {X -0.9945,Y -72.2513,Z 76,A -94.4922,B 24.9062,C -2.2361,E1 25.0026,E2 -181.1676} C_DIS
Enddeposition()
LIN {X 0.4617,Y -71.2706,Z 76,A -93.7337,B 24.9057,C -2.2425,E1 25.0047,E2 -181.9413} C_DIS
Startdeposition()
$VEL.CP = VEL_PRINT
LIN {X -1.5902,Y -71.2653,Z 76,A -97.3273,B 24.9099,C -2.1921,E1 24.9944,E2 -178.2279} C_DIS
LIN {X -5.2108,Y -71.0925,Z 76,A -100.0026,B 24.9094,C -2.1979,E1 24.9869,E2 -175.5657} C_DIS
LIN {X -9.7588,Y -70.6118,Z 76,A -103.5316,B 24.909,C -2.2021,E1 24.9772,E2 -172.0443} C_DIS
LIN {X -12.2386,Y -70.2236,Z 76,A -106.6582,B 24.9112,C -2.1755,E1 24.9684,E2 -168.8514} C_DIS
LIN {X -16.203,Y -69.4167,Z 76,A -108.5652,B 24.9084,C -2.2099,E1 24.9634,E2 -167.0237} C_DIS
LIN {X -18.239,Y -68.9105,Z 76,A -110.6722,B 24.9092,C -2.2005,E1 24.9576,E2 -164.8913} C_DIS
LIN {X -21.8468,Y -67.8522,Z 76,A -114.1526,B 24.9099,C -2.1916,E1 24.9483,E2 -161.3837} C_DIS
LIN {X -25.6385,Y -66.5134,Z 76,A -116.9591,B 24.9088,C -2.2046,E1 24.941,E2 -158.6026} C_DIS
LIN {X -28.4506,Y -65.3587,Z 76,A -119.3711,B 24.9086,C -2.2079,E1 24.9348,E2 -156.1928} C_DIS
LIN {X -31.0599,Y -64.1601,Z 76,A -122.0528,B 24.9091,C -2.2017,E1 24.928,E2 -153.4895} C_DIS
LIN {X -34.5155,Y -62.3694,Z 76,A -125.3275,B 24.9091,C -2.2024,E1 24.9199,E2 -150.2071} C_DIS
LIN {X -39.5982,Y -59.2736,Z 76,A -129.6764,B 24.9076,C -2.2197,E1 24.9097,E2 -145.8856} C_DIS
LIN {X -42.1688,Y -57.4716,Z 76,A -132.4578,B 24.9077,C -2.218,E1 24.9034,E2 -143.0903} C_DIS
LIN {X -45.8493,Y -54.5818,Z 76,A -135.6286,B 24.906,C -2.2384,E1 24.8966,E2 -139.9565} C_DIS
LIN {X -47.9022,Y -52.7895,Z 76,A -138.1189,B 24.9062,C -2.2357,E1 24.8913,E2 -137.4499} C_DIS
LIN {X -50.4002,Y -50.4099,Z 76,A -140.9559,B 24.9059,C -2.24,E1 24.8856,E2 -134.6112} C_DIS
LIN {X -53.0844,Y -47.5736,Z 76,A -144.6094,B 24.9063,C -2.2352,E1 24.8787,E2 -130.9302} C_DIS
LIN {X -56.4531,Y -43.5229,Z 76,A -148.1837,B 24.9042,C -2.2599,E1 24.8725,E2 -127.3982} C_DIS
LIN {X -58.8384,Y -40.2412,Z 76,A -152.1703,B 24.9049,C -2.2517,E1 24.866,E2 -123.3725} C_DIS
LIN {X -61.2694,Y -36.4319,Z 76,A -155.7855,B 24.904,C -2.2615,E1 24.8608,E2 -119.7621} C_DIS
LIN {X -63.817,Y -31.7584,Z 76,A -159.4577,B 24.9019,C -2.2865,E1 24.856,E2 -116.1299} C_DIS
LIN {X -65.3259,Y -28.5257,Z 76,A -162.3343,B 24.9012,C -2.2943,E1 24.8527,E2 -113.2562} C_DIS
LIN {X -66.6346,Y -25.3186,Z 76,A -165.6308,B 24.9015,C -2.2911,E1 24.8493,E2 -109.9336} C_DIS
LIN {X -67.703,Y -22.3068,Z 76,A -168.2035,B 24.9009,C -2.2985,E1 24.847,E2 -107.3639} C_DIS
LIN {X -68.9825,Y -17.9626,Z 76,A -171.5348,B 24.8994,C -2.3161,E1 24.8445,E2 -104.0554} C_DIS
LIN {X -69.772,Y -14.5992,Z 76,A -174.0374,B 24.8981,C -2.3305,E1 24.843,E2 -101.5725} C_DIS
LIN {X -70.2323,Y -12.1982,Z 76,A -177.2266,B 24.8999,C -2.3102,E1 24.8415,E2 -98.3159} C_DIS
LIN {X -70.7991,Y -8.2878,Z 76,A -178.8942,B 24.8961,C -2.3526,E1 24.8409,E2 -96.7397} C_DIS
LIN {X -71.0736,Y -5.4583,Z 76,A 178.4709,B 24.8961,C -2.3521,E1 24.8402,E2 -94.0878} C_DIS
LIN {X -71.2169,Y -3.0568,Z 76,A 176.2223,B 24.8962,C -2.3514,E1 24.8399,E2 -91.8239} C_DIS
LIN {X -71.2831,Y 0.1304,Z 76,A 173.3864,B 24.8961,C -2.3537,E1 24.8399,E2 -88.9762} C_DIS
LIN {X -71.109,Y 4.9733,Z 76,A 170.2104,B 24.8936,C -2.3816,E1 24.8402,E2 -85.8478} C_DIS
LIN {X -70.7851,Y 8.4066,Z 76,A 166.9784,B 24.8936,C -2.3804,E1 24.8411,E2 -82.5937} C_DIS
LIN {X -69.9886,Y 13.5201,Z 76,A 162.3031,B 24.8935,C -2.3825,E1 24.8433,E2 -77.8956} C_DIS
LIN {X -69.112,Y 17.4589,Z 76,A 159.6418,B 24.8914,C -2.4051,E1 24.845,E2 -75.2727} C_DIS
LIN {X -68.4129,Y 20.0235,Z 76,A 157.3836,B 24.8911,C -2.4091,E1 24.8467,E2 -73.0111} C_DIS
LIN {X -67.4655,Y 23.0144,Z 76,A 154.7997,B 24.8905,C -2.4155,E1 24.849,E2 -70.4277} C_DIS
LIN {X -65.9845,Y 26.9677,Z 76,A 151.3218,B 24.8897,C -2.424,E1 24.8525,E2 -66.9504} C_DIS
LIN {X -63.5827,Y 32.2257,Z 76,A 147.13,B 24.8876,C -2.4476,E1 24.8574,E2 -62.7922} C_DIS
LIN {X -62.2284,Y 34.768,Z 76,A 144.1638,B 24.8883,C -2.4401,E1 24.8614,E2 -59.7924} C_DIS
LIN {X -60.2642,Y 38.073,Z 76,A 140.7243,B 24.8882,C -2.4411,E1 24.8665,E2 -56.3379} C_DIS
LIN {X -57.59,Y 42.0072,Z 76,A 136.8892,B 24.8872,C -2.4512,E1 24.8727,E2 -52.5081} C_DIS
LIN {X -55.103,Y 45.2222,Z 76,A 134.0837,B 24.8855,C -2.4698,E1 24.8775,E2 -49.7337} C_DIS
LIN {X -53.0344,Y 47.6294,Z 76,A 131.0533,B 24.8859,C -2.4656,E1 24.8832,E2 -46.6798} C_DIS
LIN {X -49.0944,Y 51.6823,Z 76,A 127.3306,B 24.8832,C -2.4947,E1 24.8904,E2 -43.0107} C_DIS
LIN {X -47.5947,Y 53.0655,Z 76,A 125.3686,B 24.8835,C -2.4912,E1 24.8945,E2 -41.0325} C_DIS
LIN {X -45.2215,Y 55.1033,Z 76,A 122.3175,B 24.8841,C -2.4847,E1 24.9011,E2 -37.9541} C_DIS
LIN {X -41.6908,Y 57.8196,Z 76,A 119.135,B 24.8826,C -2.501,E1 24.9081,E2 -34.7991} C_DIS
LIN {X -39.4218,Y 59.39,Z 76,A 117.0086,B 24.882,C -2.5073,E1 24.913,E2 -32.6808} C_DIS
LIN {X -36.7227,Y 61.0963,Z 76,A 114.0619,B 24.8824,C -2.5033,E1 24.9201,E2 -29.7155} C_DIS
LIN {X -33.921,Y 62.6942,Z 76,A 111.0189,B 24.8829,C -2.4975,E1 24.9276,E2 -26.6499} C_DIS
LIN {X -30.6243,Y 64.3694,Z 76,A 108.8412,B 24.8808,C -2.5203,E1 24.933,E2 -24.5209} C_DIS
LIN {X -27.7993,Y 65.6384,Z 76,A 106.2642,B 24.8806,C -2.5219,E1 24.9396,E2 -21.9415} C_DIS
LIN {X -25.128,Y 66.7068,Z 76,A 103.3891,B 24.8816,C -2.5118,E1 24.9472,E2 -19.0365} C_DIS
LIN {X -22.076,Y 67.7781,Z 76,A 101.5125,B 24.8797,C -2.5318,E1 24.952,E2 -17.2039} C_DIS
LIN {X -19.0657,Y 68.6865,Z 76,A 98.745,B 24.88,C -2.5288,E1 24.9595,E2 -14.4249} C_DIS
LIN {X -16.593,Y 69.3245,Z 76,A 96.4684,B 24.8803,C -2.5255,E1 24.9657,E2 -12.1371} C_DIS
LIN {X -13.0468,Y 70.0794,Z 76,A 94.0771,B 24.8789,C -2.5403,E1 24.9721,E2 -9.7783} C_DIS
LIN {X -10.0248,Y 70.5741,Z 76,A 91.28,B 24.8795,C -2.5339,E1 24.9799,E2 -6.9636} C_DIS
LIN {X -7.0427,Y 70.9348,Z 76,A 89.1903,B 24.8786,C -2.543,E1 24.9857,E2 -4.8943} C_DIS
LIN {X -4.1219,Y 71.1634,Z 76,A 86.1006,B 24.8802,C -2.5262,E1 24.9944,E2 -1.7635} C_DIS
LIN {X 1.5884,Y 71.2644,Z 76,A 81.8436,B 24.8793,C -2.5352,E1 25.0062,E2 2.4718} C_DIS
LIN {X 6.2917,Y 71.0048,Z 76,A 78.3538,B 24.8787,C -2.5424,E1 25.0159,E2 5.9429} C_DIS
LIN {X 9.7012,Y 70.619,Z 76,A 74.8165,B 24.8806,C -2.5225,E1 25.0258,E2 9.5245} C_DIS
LIN {X 13.1429,Y 70.0612,Z 76,A 73.0639,B 24.8781,C -2.5477,E1 25.0304,E2 11.2154} C_DIS
LIN {X 15.3218,Y 69.6165,Z 76,A 70.9622,B 24.879,C -2.539,E1 25.0362,E2 13.3352} C_DIS
LIN {X 19.0064,Y 68.7031,Z 76,A 67.4586,B 24.8803,C -2.5257,E1 25.0458,E2 16.865} C_DIS
LIN {X 22.4798,Y 67.6458,Z 76,A 64.9875,B 24.8794,C -2.5348,E1 25.0523,E2 19.3099} C_DIS
LIN {X 25.4095,Y 66.6002,Z 76,A 62.5349,B 24.8794,C -2.5337,E1 25.0587,E2 21.7598} C_DIS
LIN {X 27.732,Y 65.6668,Z 76,A 60.492,B 24.8798,C -2.5308,E1 25.064,E2 23.8049} C_DIS
LIN {X 30.77,Y 64.2994,Z 76,A 58.315,B 24.8788,C -2.5408,E1 25.0694,E2 25.9527} C_DIS
LIN {X 33.0528,Y 63.1555,Z 76,A 55.5905,B 24.8807,C -2.5207,E1 25.0763,E2 28.7175} C_DIS
LIN {X 36.7821,Y 61.0602,Z 76,A 52.7143,B 24.8798,C -2.5306,E1 25.0832,E2 31.5616} C_DIS
LIN {X 38.6325,Y 59.9062,Z 76,A 50.6506,B 24.8808,C -2.5197,E1 25.0881,E2 33.6444} C_DIS
LIN {X 41.0468,Y 58.2797,Z 76,A 47.687,B 24.8827,C -2.4994,E1 25.095,E2 36.6459} C_DIS
LIN {X 43.768,Y 56.2642,Z 76,A 45.3742,B 24.8822,C -2.5053,E1 25.1001,E2 38.9361} C_DIS
LIN {X 47.2219,Y 53.3985,Z 76,A 41.5477,B 24.8834,C -2.4926,E1 25.1082,E2 42.7779} C_DIS
LIN {X 49.7459,Y 51.0557,Z 76,A 39.4352,B 24.8823,C -2.5046,E1 25.1124,E2 44.8533} C_DIS
LIN {X 52.1321,Y 48.6161,Z 76,A 36.0876,B 24.8843,C -2.4824,E1 25.1189,E2 48.239} C_DIS
LIN {X 54.7154,Y 45.6886,Z 76,A 32.5174,B 24.8861,C -2.4635,E1 25.1254,E2 51.8374} C_DIS
LIN {X 57.0393,Y 42.7518,Z 76,A 30.9972,B 24.883,C -2.4969,E1 25.1279,E2 53.2714} C_DIS
LIN {X 59.3002,Y 39.5579,Z 76,A 27.5219,B 24.8846,C -2.48,E1 25.1335,E2 56.7699} C_DIS
LIN {X 62.5429,Y 34.2,Z 76,A 22.3927,B 24.886,C -2.4642,E1 25.1408,E2 61.9101} C_DIS
LIN {X 63.8289,Y 31.7345,Z 76,A 19.8727,B 24.8873,C -2.4502,E1 25.144,E2 64.4498} C_DIS
LIN {X 65.3464,Y 28.4788,Z 76,A 16.6155,B 24.889,C -2.4319,E1 25.1478,E2 67.7327} C_DIS
LIN {X 66.6976,Y 25.1521,Z 76,A 14.3043,B 24.8883,C -2.4395,E1 25.1501,E2 70.0129} C_DIS
LIN {X 67.6658,Y 22.4204,Z 76,A 11.4538,B 24.8903,C -2.4181,E1 25.1527,E2 72.8978} C_DIS
LIN {X 69.0257,Y 17.7946,Z 76,A 8.2839,B 24.8895,C -2.4262,E1 25.155,E2 76.0304} C_DIS
LIN {X 69.6271,Y 15.2729,Z 76,A 4.9342,B 24.8933,C -2.3846,E1 25.1571,E2 79.459} C_DIS
LIN {X 70.4434,Y 10.9047,Z 76,A 2.6442,B 24.8911,C -2.4093,E1 25.1581,E2 81.6772} C_DIS
LIN {X 70.6855,Y 9.206,Z 76,A 0.7716,B 24.8927,C -2.3911,E1 25.1588,E2 83.5817} C_DIS
LIN {X 71.1104,Y 4.9529,Z 76,A -2.3704,B 24.8929,C -2.3886,E1 25.1595,E2 86.7111} C_DIS
LIN {X 71.2783,Y 0.881,Z 76,A -5.6774,B 24.8939,C -2.3773,E1 25.1598,E2 90.025} C_DIS
LIN {X 71.1209,Y -4.7963,Z 76,A -9.8351,B 24.8942,C -2.3743,E1 25.1594,E2 94.1651} C_DIS
LIN {X 70.8028,Y -8.2562,Z 76,A -13.2633,B 24.8966,C -2.3475,E1 25.1584,E2 97.6363} C_DIS
LIN {X 70.1776,Y -12.502,Z 76,A -16.8649,B 24.8979,C -2.3323,E1 25.1567,E2 101.2526} C_DIS
LIN {X 69.1326,Y -17.3766,Z 76,A -20.6131,B 24.8984,C -2.327,E1 25.1543,E2 104.9917} C_DIS
LIN {X 68.2529,Y -20.5629,Z 76,A -23.2019,B 24.899,C -2.3207,E1 25.1523,E2 107.5807} C_DIS
LIN {X 66.89,Y -24.6369,Z 76,A -26.7465,B 24.9001,C -2.3075,E1 25.149,E2 111.1364} C_DIS
LIN {X 65.5439,Y -28.0237,Z 76,A -29.2769,B 24.8999,C -2.3099,E1 25.1463,E2 113.6474} C_DIS
LIN {X 63.589,Y -32.2133,Z 76,A -33.109,B 24.9011,C -2.2956,E1 25.1416,E2 117.4925} C_DIS
LIN {X 61.4503,Y -36.1259,Z 76,A -36.2052,B 24.9008,C -2.299,E1 25.1374,E2 120.5646} C_DIS
LIN {X 60.2335,Y -38.1221,Z 76,A -38.3985,B 24.9021,C -2.2849,E1 25.1342,E2 122.7801} C_DIS
LIN {X 58.3061,Y -41.0085,Z 76,A -41.3647,B 24.9031,C -2.2723,E1 25.1295,E2 125.7615} C_DIS
Enddeposition()
END
